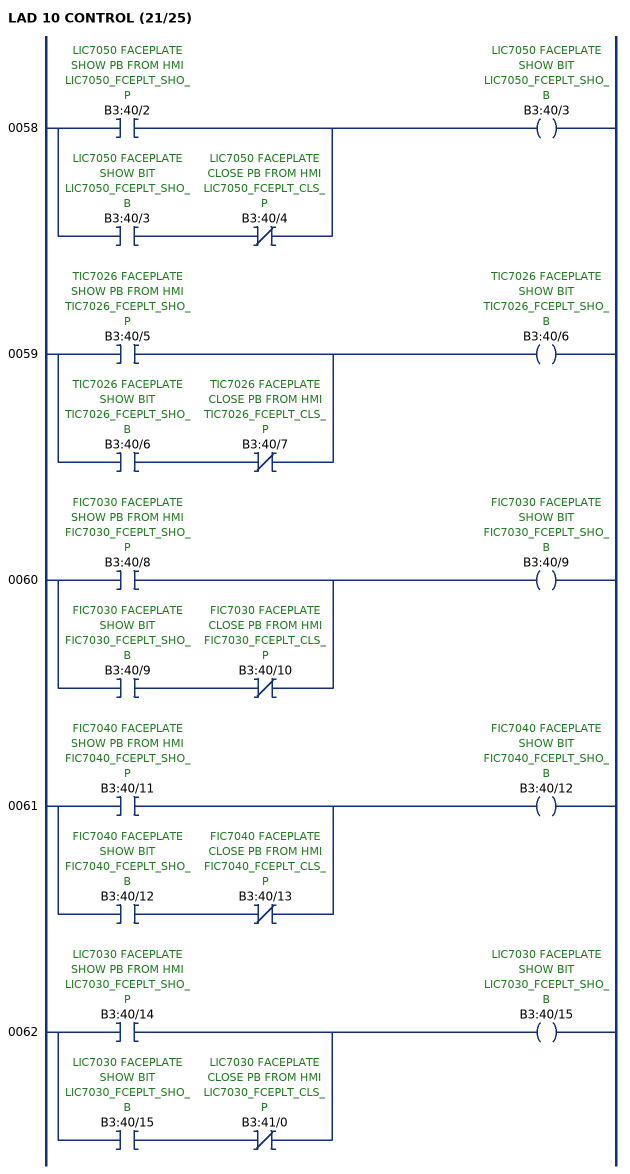
% Rung: 58 %
SOR BST XIC B3:40/2 NXB XIC B3:40/3 XIO B3:40/4 BND OTE B3:40/3 EOR
%   B3:40/2  LIC7050_FCEPLT_SHO_P  "LIC7050 FACEPLATE SHOW PB FROM HMI" %
%   B3:40/3  LIC7050_FCEPLT_SHO_B  "LIC7050 FACEPLATE SHOW BIT" %
%   B3:40/4  LIC7050_FCEPLT_CLS_P  "LIC7050 FACEPLATE CLOSE PB FROM HMI" %
% Rung: 59 %
SOR BST XIC B3:40/5 NXB XIC B3:40/6 XIO B3:40/7 BND OTE B3:40/6 EOR
%   B3:40/5  TIC7026_FCEPLT_SHO_P  "TIC7026 FACEPLATE SHOW PB FROM HMI" %
%   B3:40/6  TIC7026_FCEPLT_SHO_B  "TIC7026 FACEPLATE SHOW BIT" %
%   B3:40/7  TIC7026_FCEPLT_CLS_P  "TIC7026 FACEPLATE CLOSE PB FROM HMI" %
% Rung: 60 %
SOR BST XIC B3:40/8 NXB XIC B3:40/9 XIO B3:40/10 BND OTE B3:40/9 EOR
%   B3:40/8  FIC7030_FCEPLT_SHO_P  "FIC7030 FACEPLATE SHOW PB FROM HMI" %
%   B3:40/9  FIC7030_FCEPLT_SHO_B  "FIC7030 FACEPLATE SHOW BIT" %
%   B3:40/10  FIC7030_FCEPLT_CLS_P  "FIC7030 FACEPLATE CLOSE PB FROM HMI" %
% Rung: 61 %
SOR BST XIC B3:40/11 NXB XIC B3:40/12 XIO B3:40/13 BND OTE B3:40/12 EOR
%   B3:40/11  FIC7040_FCEPLT_SHO_P  "FIC7040 FACEPLATE SHOW PB FROM HMI" %
%   B3:40/12  FIC7040_FCEPLT_SHO_B  "FIC7040 FACEPLATE SHOW BIT" %
%   B3:40/13  FIC7040_FCEPLT_CLS_P  "FIC7040 FACEPLATE CLOSE PB FROM HMI" %
% Rung: 62 %
SOR BST XIC B3:40/14 NXB XIC B3:40/15 XIO B3:41/0 BND OTE B3:40/15 EOR
%   B3:40/14  LIC7030_FCEPLT_SHO_P  "LIC7030 FACEPLATE SHOW PB FROM HMI" %
%   B3:40/15  LIC7030_FCEPLT_SHO_B  "LIC7030 FACEPLATE SHOW BIT" %
%   B3:41/0  LIC7030_FCEPLT_CLS_P  "LIC7030 FACEPLATE CLOSE PB FROM HMI" %

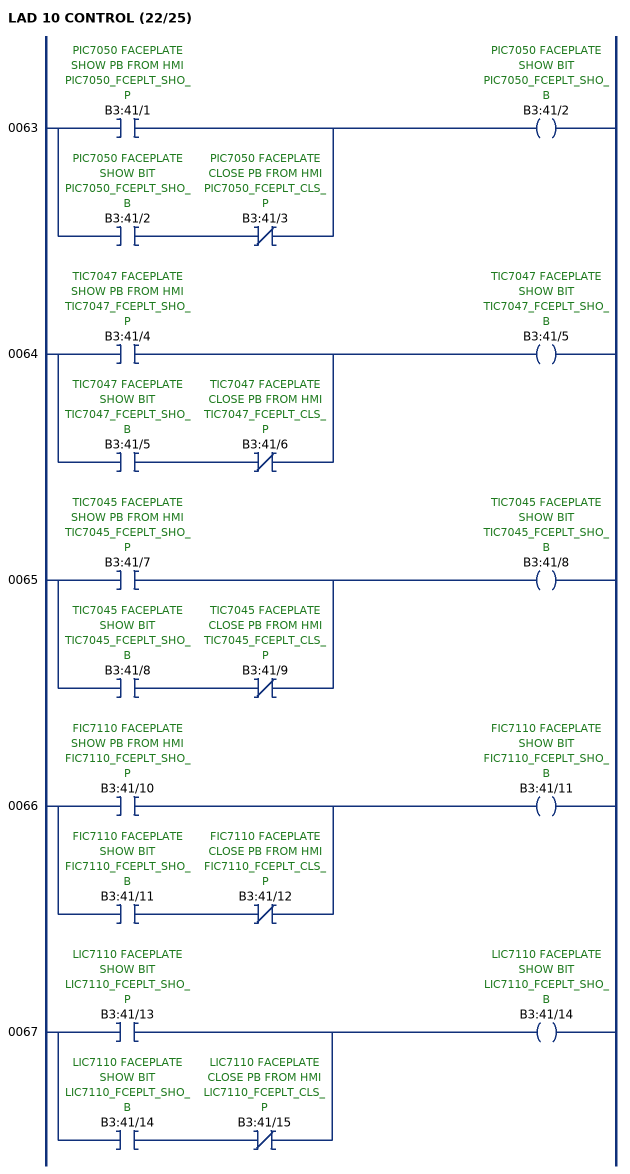
% Rung: 63 %
SOR BST XIC B3:41/1 NXB XIC B3:41/2 XIO B3:41/3 BND OTE B3:41/2 EOR
%   B3:41/1  PIC7050_FCEPLT_SHO_P  "PIC7050 FACEPLATE SHOW PB FROM HMI" %
%   B3:41/2  PIC7050_FCEPLT_SHO_B  "PIC7050 FACEPLATE SHOW BIT" %
%   B3:41/3  PIC7050_FCEPLT_CLS_P  "PIC7050 FACEPLATE CLOSE PB FROM HMI" %
% Rung: 64 %
SOR BST XIC B3:41/4 NXB XIC B3:41/5 XIO B3:41/6 BND OTE B3:41/5 EOR
%   B3:41/4  TIC7047_FCEPLT_SHO_P  "TIC7047 FACEPLATE SHOW PB FROM HMI" %
%   B3:41/5  TIC7047_FCEPLT_SHO_B  "TIC7047 FACEPLATE SHOW BIT" %
%   B3:41/6  TIC7047_FCEPLT_CLS_P  "TIC7047 FACEPLATE CLOSE PB FROM HMI" %
% Rung: 65 %
SOR BST XIC B3:41/7 NXB XIC B3:41/8 XIO B3:41/9 BND OTE B3:41/8 EOR
%   B3:41/7  TIC7045_FCEPLT_SHO_P  "TIC7045 FACEPLATE SHOW PB FROM HMI" %
%   B3:41/8  TIC7045_FCEPLT_SHO_B  "TIC7045 FACEPLATE SHOW BIT" %
%   B3:41/9  TIC7045_FCEPLT_CLS_P  "TIC7045 FACEPLATE CLOSE PB FROM HMI" %
% Rung: 66 %
SOR BST XIC B3:41/10 NXB XIC B3:41/11 XIO B3:41/12 BND OTE B3:41/11 EOR
%   B3:41/10  FIC7110_FCEPLT_SHO_P  "FIC7110 FACEPLATE SHOW PB FROM HMI" %
%   B3:41/11  FIC7110_FCEPLT_SHO_B  "FIC7110 FACEPLATE SHOW BIT" %
%   B3:41/12  FIC7110_FCEPLT_CLS_P  "FIC7110 FACEPLATE CLOSE PB FROM HMI" %
% Rung: 67 %
SOR BST XIC B3:41/13 NXB XIC B3:41/14 XIO B3:41/15 BND OTE B3:41/14 EOR
%   B3:41/13  LIC7110_FCEPLT_SHO_P  "LIC7110 FACEPLATE SHOW BIT" %
%   B3:41/14  LIC7110_FCEPLT_SHO_B  "LIC7110 FACEPLATE SHOW BIT" %
%   B3:41/15  LIC7110_FCEPLT_CLS_P  "LIC7110 FACEPLATE CLOSE PB FROM HMI" %

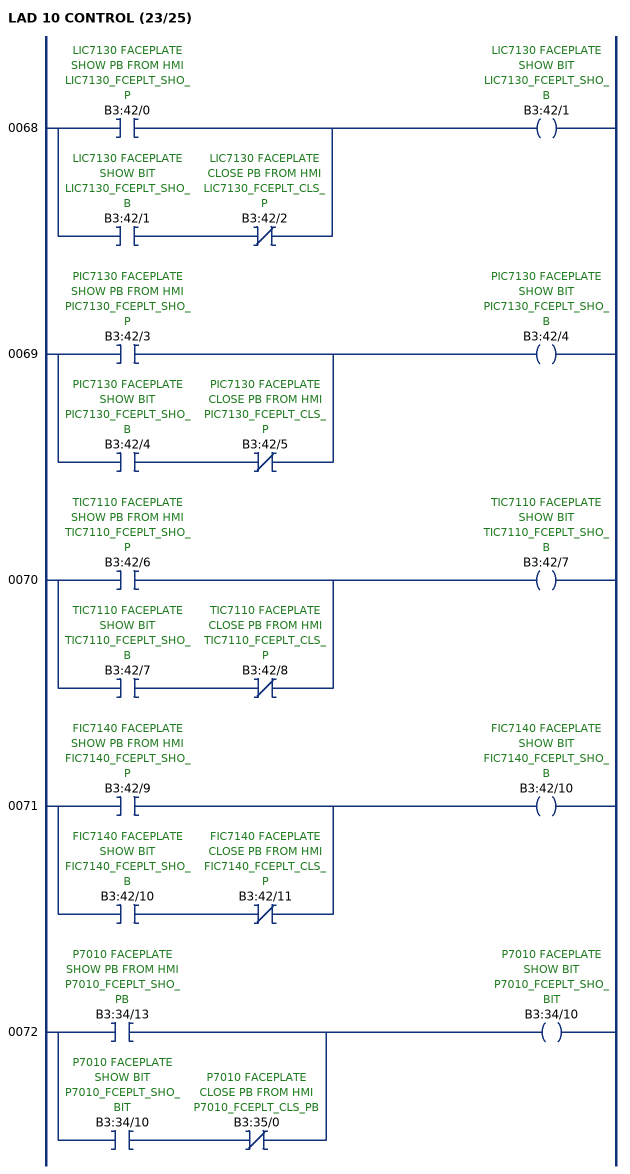
% Rung: 68 %
SOR BST XIC B3:42/0 NXB XIC B3:42/1 XIO B3:42/2 BND OTE B3:42/1 EOR
%   B3:42/0  LIC7130_FCEPLT_SHO_P  "LIC7130 FACEPLATE SHOW PB FROM HMI" %
%   B3:42/1  LIC7130_FCEPLT_SHO_B  "LIC7130 FACEPLATE SHOW BIT" %
%   B3:42/2  LIC7130_FCEPLT_CLS_P  "LIC7130 FACEPLATE CLOSE PB FROM HMI" %
% Rung: 69 %
SOR BST XIC B3:42/3 NXB XIC B3:42/4 XIO B3:42/5 BND OTE B3:42/4 EOR
%   B3:42/3  PIC7130_FCEPLT_SHO_P  "PIC7130 FACEPLATE SHOW PB FROM HMI" %
%   B3:42/4  PIC7130_FCEPLT_SHO_B  "PIC7130 FACEPLATE SHOW BIT" %
%   B3:42/5  PIC7130_FCEPLT_CLS_P  "PIC7130 FACEPLATE CLOSE PB FROM HMI" %
% Rung: 70 %
SOR BST XIC B3:42/6 NXB XIC B3:42/7 XIO B3:42/8 BND OTE B3:42/7 EOR
%   B3:42/6  TIC7110_FCEPLT_SHO_P  "TIC7110 FACEPLATE SHOW PB FROM HMI" %
%   B3:42/7  TIC7110_FCEPLT_SHO_B  "TIC7110 FACEPLATE SHOW BIT" %
%   B3:42/8  TIC7110_FCEPLT_CLS_P  "TIC7110 FACEPLATE CLOSE PB FROM HMI" %
% Rung: 71 %
SOR BST XIC B3:42/9 NXB XIC B3:42/10 XIO B3:42/11 BND OTE B3:42/10 EOR
%   B3:42/9  FIC7140_FCEPLT_SHO_P  "FIC7140 FACEPLATE SHOW PB FROM HMI" %
%   B3:42/10  FIC7140_FCEPLT_SHO_B  "FIC7140 FACEPLATE SHOW BIT" %
%   B3:42/11  FIC7140_FCEPLT_CLS_P  "FIC7140 FACEPLATE CLOSE PB FROM HMI" %
% Rung: 72 %
SOR BST XIC B3:34/13 NXB XIC B3:34/10 XIO B3:35/0 BND OTE B3:34/10 EOR
%   B3:34/13  P7010_FCEPLT_SHO_PB  "P7010 FACEPLATE SHOW PB FROM HMI" %
%   B3:34/10  P7010_FCEPLT_SHO_BIT  "P7010 FACEPLATE SHOW BIT" %
%   B3:35/0  P7010_FCEPLT_CLS_PB  "P7010 FACEPLATE CLOSE PB FROM HMI" %

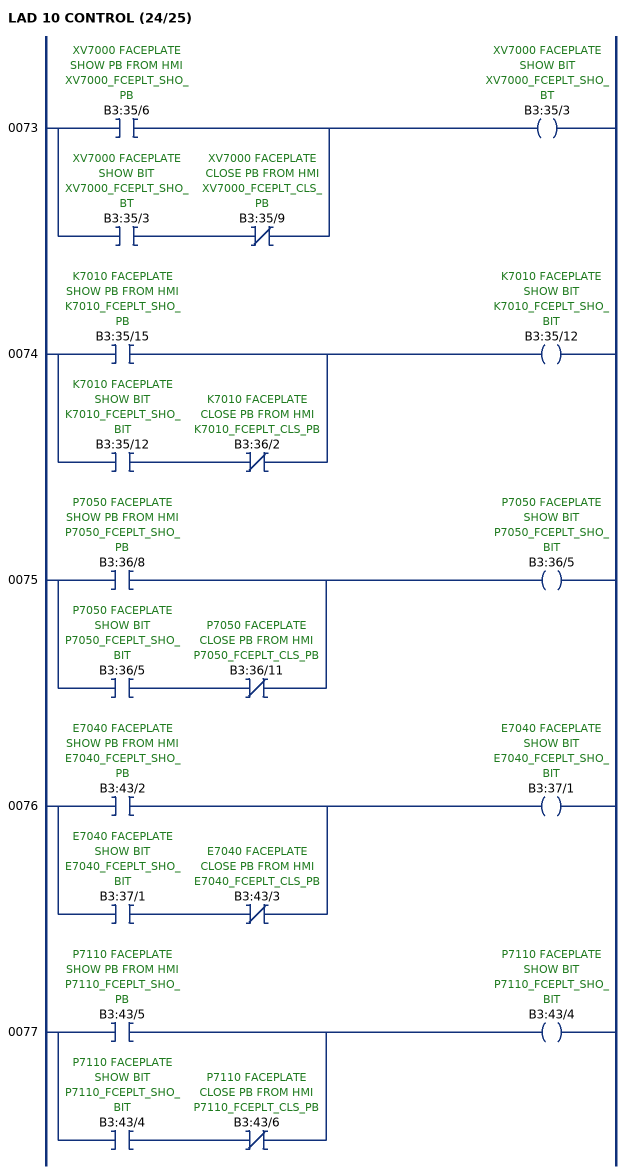
% Rung: 73 %
SOR BST XIC B3:35/6 NXB XIC B3:35/3 XIO B3:35/9 BND OTE B3:35/3 EOR
%   B3:35/6  XV7000_FCEPLT_SHO_PB  "XV7000 FACEPLATE SHOW PB FROM HMI" %
%   B3:35/3  XV7000_FCEPLT_SHO_BT  "XV7000 FACEPLATE SHOW BIT" %
%   B3:35/9  XV7000_FCEPLT_CLS_PB  "XV7000 FACEPLATE CLOSE PB FROM HMI" %
% Rung: 74 %
SOR BST XIC B3:35/15 NXB XIC B3:35/12 XIO B3:36/2 BND OTE B3:35/12 EOR
%   B3:35/15  K7010_FCEPLT_SHO_PB  "K7010 FACEPLATE SHOW PB FROM HMI" %
%   B3:35/12  K7010_FCEPLT_SHO_BIT  "K7010 FACEPLATE SHOW BIT" %
%   B3:36/2  K7010_FCEPLT_CLS_PB  "K7010 FACEPLATE CLOSE PB FROM HMI" %
% Rung: 75 %
SOR BST XIC B3:36/8 NXB XIC B3:36/5 XIO B3:36/11 BND OTE B3:36/5 EOR
%   B3:36/8  P7050_FCEPLT_SHO_PB  "P7050 FACEPLATE SHOW PB FROM HMI" %
%   B3:36/5  P7050_FCEPLT_SHO_BIT  "P7050 FACEPLATE SHOW BIT" %
%   B3:36/11  P7050_FCEPLT_CLS_PB  "P7050 FACEPLATE CLOSE PB FROM HMI" %
% Rung: 76 %
SOR BST XIC B3:43/2 NXB XIC B3:37/1 XIO B3:43/3 BND OTE B3:37/1 EOR
%   B3:43/2  E7040_FCEPLT_SHO_PB  "E7040 FACEPLATE SHOW PB FROM HMI" %
%   B3:37/1  E7040_FCEPLT_SHO_BIT  "E7040 FACEPLATE SHOW BIT" %
%   B3:43/3  E7040_FCEPLT_CLS_PB  "E7040 FACEPLATE CLOSE PB FROM HMI" %
% Rung: 77 %
SOR BST XIC B3:43/5 NXB XIC B3:43/4 XIO B3:43/6 BND OTE B3:43/4 EOR
%   B3:43/5  P7110_FCEPLT_SHO_PB  "P7110 FACEPLATE SHOW PB FROM HMI" %
%   B3:43/4  P7110_FCEPLT_SHO_BIT  "P7110 FACEPLATE SHOW BIT" %
%   B3:43/6  P7110_FCEPLT_CLS_PB  "P7110 FACEPLATE CLOSE PB FROM HMI" %

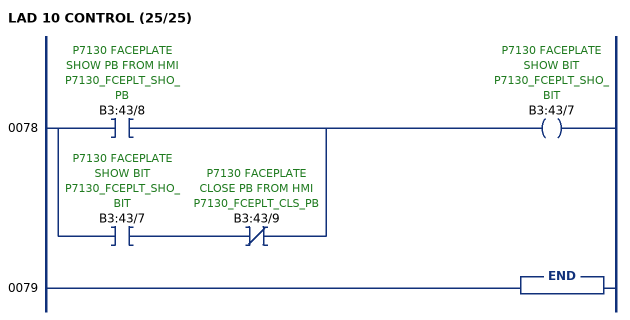
% Rung: 78 %
SOR BST XIC B3:43/8 NXB XIC B3:43/7 XIO B3:43/9 BND OTE B3:43/7 EOR
%   B3:43/8  P7130_FCEPLT_SHO_PB  "P7130 FACEPLATE SHOW PB FROM HMI" %
%   B3:43/7  P7130_FCEPLT_SHO_BIT  "P7130 FACEPLATE SHOW BIT" %
%   B3:43/9  P7130_FCEPLT_CLS_PB  "P7130 FACEPLATE CLOSE PB FROM HMI" %
% Rung: 79 %
SOR END EOR

OTHER DOCUMENTED ADDRESSES
  B3:46/11  "DUMMY"
  B3:47/0  "ONE SHOT"
  B3:47/1  "ONE SHOT"
  B3:47/2  "ONE SHOT"
  B3:47/3  "ONE SHOT"
  B3:47/4  "ONE SHOT"
  B3:47/5  "ONE SHOT"
  B3:47/6  "ONE SHOT"
  B3:47/7  "ONE SHOT"
  B3:47/8  "ONE SHOT"
  B3:47/9  "ONE SHOT"
  B3:47/10  "ONE SHOT"
  B3:47/11  "ONE SHOT"
  B3:47/12  "ONE SHOT"
  B3:47/13  "ONE SHOT"
  B3:47/14  "ONE SHOT"
  B3:47/15  "ONE SHOT"
  B3:48/0  "ONE SHOT"
  B3:48/1  "ONE SHOT"
  B3:48/2  "ONE SHOT"
  B9:36/2  "ESD LIC-7130 OFF"
  DFILE:0  "OUTPUT"
  DFILE:1  "INPUT"
  DFILE:2  "STATUS"
  DFILE:3  "BINARY"
  DFILE:4  "TIMER"
  DFILE:5  "COUNTER"
  DFILE:6  "CONTROL"
  DFILE:7  "INTEGER"
  DFILE:8  "FLOAT"
  DFILE:9  "ALARMS"
  DFILE:10  "F-SETPTS 1"
  DFILE:11  "N-SETPTS 1"
  DFILE:12  "PIDBLOCKS1"
  DFILE:13  "DONOTTOUCH"
  DFILE:14  "PIDBLOCKS2"
  DFILE:15  "PIDBLOCKS3"
  DFILE:16  "SYSCTRLS"
  DFILE:17  "TIMERS 2"
  DFILE:18  "F-SETPTS 2"
  DFILE:19  "N-SETPTS 2"
  DFILE:20  "MB_CFG"
  DFILE:21  "MB_BIN"
  DFILE:22  "MB_FLT1"
  DFILE:23  "MB_FLT2"
  DFILE:24  "MB_FLT3"
  DFILE:25  "MB_FLT4"
  DFILE:26  "MB_FLT5"
  DFILE:27  "MB_FLT6"
  DFILE:28  "MB_FLT7"
  DFILE:29  "COMP_4"
  F10:[N7:100]  F18
  F22:0  FT_7002_SCI_PLC  "FT-7002 Scaled In 0-600 PLC -> DeltaV"
  F22:1  FT_7010_SCI_PLC  "FT-7010 Scaled In 0-200 PLC -> DeltaV"
  F22:2  LT_7010_SCI_PLC  "LT-7010 Scaled In 0-100 PLC -> DeltaV"
  F22:3  PT_7010_SCI_PLC  "PT-7010 Scaled In 0-200 PLC -> DeltaV"
  F22:4  PT_7020_SCI_PLC  "PT-7020 Scaled In 0-1000 PLC -> DeltaV"
  F22:5  FT_7000_SCI_PLC  "FT-7000 Scaled In 0-40 PLC -> DeltaV"
  F22:6  FT_7005_SCI_PLC  "FT-7005 Scaled In 0-300 PLC -> DeltaV"
  F22:7  FT_7008_SCI_PLC  "FT-7008 Scaled In 0-500 PLC -> DeltaV"
  F22:8  FT_7025_SCI_PLC  "FT-7025 Scaled In 0-200 PLC -> DeltaV"
  F22:9  FT_7050_SCI_PLC  "FT-7050 Scaled In 0-150 PLC -> DeltaV"
  F22:10  LT_7050_SCI_PLC  "LT-7050 Scaled In 0-100 PLC -> DeltaV"
  F22:11  PT_7000_SCI_PLC  "PT-7000 Scaled In 0-1000 PLC -> DeltaV"
  F22:12  PT_7015_SCI_PLC  "PT-7015 Scaled In 0-1000 PLC -> DeltaV"
  F22:13  PT_7025_SCI_PLC  "PT-7025 Scaled In 0-1000 PLC -> DeltaV"
  F22:14  FT_7030_SCI_PLC  "FT-7030 Scaled In 0-200 PLC -> DeltaV"
  F22:15  FT_7040_SCI_PLC  "FT-7040 Scaled In 0-50 PLC -> DeltaV"
  F22:16  FT_7052_SCI_PLC  "FT-7052 Scaled In 0-150 PLC -> DeltaV"
  F22:17  LT_7030_SCI_PLC  "LT-7030 Scaled In 0-100 PLC -> DeltaV"
  F22:18  PDT_7040_SCI_PLC  "PDT-7040 Scaled In 0-5 PLC -> DeltaV"
  F22:19  PT_7030_SCI_PLC  "PT-7030 Scaled In 0-1000 PLC -> DeltaV"
  F22:20  PT_7040_SCI_PLC  "PT-7040 Scaled In 0-1000 PLC -> DeltaV"
  F22:21  PT_7050_SCI_PLC  "PT-7050 Scaled In 0-1000 PLC -> DeltaV"
  F22:22  ST_7040_SCI_PLC  "ST-7040 Scaled In 0-100 PLC -> DeltaV"
  F22:23  FT_7095_SCI_PLC  "FT-7095 Scaled In 0-700 PLC -> DeltaV"
  F22:24  FT_7110_SCI_PLC  "FT-7110 Scaled In 0-400 PLC -> DeltaV"
  F22:25  FT_7130_SCI_PLC  "FT-7130 Scaled In 0-3 PLC -> DeltaV"
  F22:26  FT_7132_SCI_PLC  "FT-7132 Scaled In 0-700 PLC -> DeltaV"
  F22:27  FT_7145_SCI_PLC  "FT-7145 Scaled In 0-400 PLC -> DeltaV"
  F22:28  LT_7110_SCI_PLC  "LT-7110 Scaled In 0-100 PLC -> DeltaV"
  F22:29  LT_7130_SCI_PLC  "LT-7130 Scaled In 0-100 PLC -> DeltaV"
  F22:30  PDT_7110_SCI_PLC  "PDT-7110 Scaled In 0-5 PLC -> DeltaV"
  F22:31  PT_7110_SCI_PLC  "PT-7110 Scaled In 0-300 PLC -> DeltaV"
  F22:32  PT_7111_SCI_PLC  "PT-7111 Scaled In 0-200 PLC -> DeltaV"
  F22:33  PT_7130_SCI_PLC  "PT-7130 Scaled In 0-200 PLC -> DeltaV"
  F22:34  ST_7110_SCI_PLC  "ST-7110 Scaled In 0-100 PLC -> DeltaV"
  F22:35  ST_7130_SCI_PLC  "ST-7130 Scaled In 0-100 PLC -> DeltaV"
  F22:36  FT_7120_SCI_PLC  "FT-7120 Scaled In 0-400 PLC -> DeltaV"
  F22:37  FT_7140_SCI_PLC  "FT-7140 Scaled In (-454-2498) PLC -> DeltaV"
  F22:38  TT_7009_SCI_PLC  "TT-7009 Scaled In (-454-2498) PLC -> DeltaV"
  F22:39  TT_7010_SCI_PLC  "TT-7010 Scaled In (-454-2498) PLC -> DeltaV"
  F22:40  TT_7020_SCI_PLC  "TT-7020 Scaled In (-454-2498) PLC -> DeltaV"
  F22:41  TT_7000_SCI_PLC  "TT-7000 Scaled In (-454-2498) PLC -> DeltaV"
  F22:42  TT_7015_SCI_PLC  "TT-7015 Scaled In (-454-2498) PLC -> DeltaV"
  F22:43  TT_7025_SCI_PLC  "TT-7025 Scaled In (-454-2498) PLC -> DeltaV"
  F22:44  TT_7026_SCI_PLC  "TT-7026 Scaled In (-454-2498) PLC -> DeltaV"
  F22:45  TT_7050_SCI_PLC  "TT-7050 Scaled In (-454-2498) PLC -> DeltaV"
  F22:46  TT_7030_SCI_PLC  "TT-7030 Scaled In (-454-2498) PLC -> DeltaV"
  F22:47  TT_7040_SCI_PLC  "TT-7040 Scaled In (-454-2498) PLC -> DeltaV"
  F22:48  TT_7042_SCI_PLC  "TT-7042 Scaled In (-454-2498) PLC -> DeltaV"
  F22:49  TT_7043_SCI_PLC  "TT-7043 Scaled In (-454-2498) PLC -> DeltaV"
  F22:50  TT_7044_SCI_PLC  "TT-7044 Scaled In (-454-2498) PLC -> DeltaV"
  F22:51  TT_7045_SCI_PLC  "TT-7045 Scaled In (-454-2498) PLC -> DeltaV"
  F22:52  TT_7046_SCI_PLC  "TT-7046 Scaled In (-454-2498) PLC -> DeltaV"
  F22:53  TT_7047_SCI_PLC  "TT-7047 Scaled In (-454-2498) PLC -> DeltaV"
  F22:54  TT_7110_SCI_PLC  "TT-7110 Scaled In (-454-2498) PLC -> DeltaV"
  F22:55  TT_7111_SCI_PLC  "TT-7111 Scaled In (-454-2498) PLC -> DeltaV"
  F22:56  TT_7118_SCI_PLC  "TT-7118 Scaled In (-454-2498) PLC -> DeltaV"
  F22:57  TT_7119_SCI_PLC  "TT-7119 Scaled In (-454-2498) PLC -> DeltaV"
  F22:58  TT_7130_SCI_PLC  "TT-7130 Scaled In (-454-2498) PLC -> DeltaV"
  F22:59  ST_7010_SCI_PLC  "ST-7010 Scaled In 0-100 PLC -> DeltaV"
  F22:60  TT_7135_SCI_PLC  "TT-7135 Scaled In (-454-2498) PLC -> DeltaV"
  F22:61  TT_7140_SCI_PLC  "TT-7140 Scaled In (-454-2498) PLC -> DeltaV"
  F22:62  TT_7145_SCI_PLC  "TT-7145 Scaled In (-454-2498) PLC -> DeltaV"
  F22:63  PT_7026_SCI_PLC  "PT-7026 Scaled In 0-1000 PLC -> DeltaV"
  F22:64  TT_7027_SCI_PLC  "TT-7027 Scaled In (-454-2498) PLC -> DeltaV"
  F22:65  FIC7015_PV_PLC  "FIC7015 PV SCALED FOR HMI PLC -> DeltaV"
  F22:66  TIC7010_PV_PLC  "TIC7010 PV SCALED FOR HMI PLC -> DeltaV"
  F22:67  FIC7000_PV_PLC  "FIC7000 PV SCALED FOR HMI PLC -> DeltaV"
  F22:68  FIC7005_PV_PLC  "FIC7005 PV SCALED FOR HMI PLC -> DeltaV"
  F22:69  FIC7008_PV_PLC  "FIC7008 PV SCALED FOR HMI PLC -> DeltaV"
  F22:70  FIC7010_PV_PLC  "FIC7010 PV SCALED FOR HMI PLC -> DeltaV"
  F22:71  LIC7050_PV_PLC  "LIC7050 PV SCALED FOR HMI PLC -> DeltaV"
  F22:72  TIC7026_PV_PLC  "TIC7026 PV SCALED FOR HMI PLC -> DeltaV"
  F22:73  FIC7030_PV_PLC  "FIC7030 PV SCALED FOR HMI PLC -> DeltaV"
  F22:74  FIC7040_PV_PLC  "FIC7040 PV SCALED FOR HMI PLC -> DeltaV"
  F22:75  LIC7030_PV_PLC  "LIC7030 PV SCALED FOR HMI PLC -> DeltaV"
  F22:76  PIC7050_PV_PLC  "PIC7050 PV SCALED FOR HMI PLC -> DeltaV"
  F22:77  TIC7047_PV_PLC  "TIC7047 PV SCALED FOR HMI PLC -> DeltaV"
  F22:78  TIC7045_PV_PLC  "TIC7045 PV SCALED FOR HMI PLC -> DeltaV"
  F22:79  FIC7110_PV_PLC  "FIC7110 PV SCALED FOR HMI PLC -> DeltaV"
  F22:80  LIC7110_PV_PLC  "LIC7110 PV SCALED FOR HMI PLC -> DeltaV"
  F22:81  LIC7130_PV_PLC  "LIC7130 PV SCALED FOR HMI PLC -> DeltaV"
  F22:82  PIC7130_PV_PLC  "PIC7130 PV SCALED FOR HMI PLC -> DeltaV"
  F22:83  TIC7110_PV_PLC  "TIC7110 PV SCALED FOR HMI PLC -> DeltaV"
  F22:84  FIC7140_PV_PLC  "FIC7140 PV SCALED FOR HMI PLC -> DeltaV"
  F22:85  WATCHDOG_TIMER_PLC  "PLC WATCHDOG TIMER PLC -> DeltaV"
  F23:0  FT_7002_L_AL_SP_PLC  "FT-7002 LO ALARM SP PLC -> DeltaV"
  F23:1  FT_7002_H_AL_SP_PLC  "FT-7002 HI ALARM SP PLC -> DeltaV"
  F23:2  FT_7010_L_AL_SP_PLC  "FT-7010 LO ALARM SP PLC -> DeltaV"
  F23:3  FT_7010_H_AL_SP_PLC  "FT-7010 HI ALARM SP PLC -> DeltaV"
  F23:4  LT_7010_L_AL_SP_PLC  "LT-7010 LO ALARM SP PLC -> DeltaV"
  F23:5  LT_7010_H_AL_SP_PLC  "LT-7010 HI ALARM SP PLC -> DeltaV"
  F23:6  PT_7010_L_AL_SP_PLC  "PT-7010 LO ALARM SP PLC -> DeltaV"
  F23:7  PT_7010_H_AL_SP_PLC  "PT-7010 HI ALARM SP PLC -> DeltaV"
  F23:8  PT_7020_L_AL_SP_PLC  "PT-7020 LO ALARM SP PLC -> DeltaV"
  F23:9  PT_7020_H_AL_SP_PLC  "PT-7020 HI ALARM SP PLC -> DeltaV"
  F23:10  FT_7000_L_AL_SP_PLC  "FT-7000 LO ALARM SP PLC -> DeltaV"
  F23:11  FT_7000_H_AL_SP_PLC  "FT-7000 HI ALARM SP PLC -> DeltaV"
  F23:12  FT_7005_L_AL_SP_PLC  "FT-7005 LO ALARM SP PLC -> DeltaV"
  F23:13  FT_7005_H_AL_SP_PLC  "FT-7005 HI ALARM SP PLC -> DeltaV"
  F23:14  FT_7008_L_AL_SP_PLC  "FT-7008 LO ALARM SP PLC -> DeltaV"
  F23:15  FT_7008_H_AL_SP_PLC  "FT-7008 HI ALARM SP PLC -> DeltaV"
  F23:16  FT_7025_L_AL_SP_PLC  "FT-7025 LO ALARM SP PLC -> DeltaV"
  F23:17  FT_7025_H_AL_SP_PLC  "FT-7025 HI ALARM SP PLC -> DeltaV"
  F23:18  FT_7050_L_AL_SP_PLC  "FT-7050 LO ALARM SP PLC -> DeltaV"
  F23:19  FT_7050_H_AL_SP_PLC  "FT-7050 HI ALARM SP PLC -> DeltaV"
  F23:20  LT_7050_L_AL_SP_PLC  "LT-7050 LO ALARM SP PLC -> DeltaV"
  F23:21  LT_7050_H_AL_SP_PLC  "LT-7050 HI ALARM SP PLC -> DeltaV"
  F23:22  PT_7000_L_AL_SP_PLC  "PT-7000 LO ALARM SP PLC -> DeltaV"
  F23:23  PT_7000_H_AL_SP_PLC  "PT-7000 HI ALARM SP PLC -> DeltaV"
  F23:24  PT_7015_L_AL_SP_PLC  "PT-7015 LO ALARM SP PLC -> DeltaV"
  F23:25  PT_7015_H_AL_SP_PLC  "PT-7015 HI ALARM SP PLC -> DeltaV"
  F23:26  PT_7025_L_AL_SP_PLC  "PT-7025 LO ALARM SP PLC -> DeltaV"
  F23:27  PT_7025_H_AL_SP_PLC  "PT-7025 HI ALARM SP PLC -> DeltaV"
  F23:28  FT_7030_L_AL_SP_PLC  "FT-7030 LO ALARM SP PLC -> DeltaV"
  F23:29  FT_7030_H_AL_SP_PLC  "FT-7030 HI ALARM SP PLC -> DeltaV"
  F23:30  FT_7040_L_ALSP_PLC  "FT-7040 LO ALARM SP PLC -> DeltaV"
  F23:31  FT_7040_H_AL_SP_PLC  "FT-7040 HI ALARM SP PLC -> DeltaV"
  F23:32  FT_7052_L_AL_SP_PLC  "FT-7052 LO ALARM SP PLC -> DeltaV"
  F23:33  FT_7052_H_AL_SP_PLC  "FT-7052 HI ALARM SP PLC -> DeltaV"
  F23:34  LT_7030_L_AL_SP_PLC  "LT-7030 LO ALARM SP PLC -> DeltaV"
  F23:35  LT_7030_H_AL_SP_PLC  "LT-7030 HI ALARM SP PLC -> DeltaV"
  F23:36  PDT_7040_L_AL_SP_PLC  "PDT-7040 LO ALARM SP PLC -> DeltaV"
  F23:37  PDT_7040_H_AL_SP_PLC  "PDT-7040 HI ALARM SP PLC -> DeltaV"
  F23:38  PT_7030_L_AL_SP_PLC  "PT-7030 LO ALARM SP PLC -> DeltaV"
  F23:39  PT_7030_H_AL_SP_PLC  "PT-7030 HI ALARM SP PLC -> DeltaV"
  F23:40  PT_7040_L_AL_SP_PLC  "PT-7040 LO ALARM SP PLC -> DeltaV"
  F23:41  PT_7040_H_AL_SP_PLC  "PT-7040 HI ALARM SP PLC -> DeltaV"
  F23:42  PT_7050_L_AL_SP_PLC  "PT-7050 LO ALARM SP PLC -> DeltaV"
  F23:43  PT_7050_H_AL_SP_PLC  "PT-7050 HI ALARM SP PLC -> DeltaV"
  F23:44  ST_7040_L_AL_SP_PLC  "ST-7040 LO ALARM SP PLC -> DeltaV"
  F23:45  ST_7040_H_AL_SP_PLC  "ST-7040 HI ALARM SP PLC -> DeltaV"
  F23:46  FT_7095_L_AL_SP_PLC  "FT-7095 LO ALARM SP PLC -> DeltaV"
  F23:47  FT_7095_H_AL_SP_PLC  "FT-7095 HI ALARM SP PLC -> DeltaV"
  F23:48  FT_7110_L_AL_SP_PLC  "FT-7110 LO ALARM SP PLC -> DeltaV"
  F23:49  FT_7110_H_AL_SP_PLC  "FT-7110 HI ALARM SP PLC -> DeltaV"
  F23:50  FT_7130_L_AL_SP_PLC  "FT-7130 LO ALARM SP PLC -> DeltaV"
  F23:51  FT_7130_H_AL_SP_PLC  "FT-7130 HI ALARM SP PLC -> DeltaV"
  F23:52  FT_7132_L_AL_SP_PLC  "FT-7132 LO ALARM SP PLC -> DeltaV"
  F23:53  FT_7132_H_AL_SP_PLC  "FT-7132 HI ALARM SP PLC -> DeltaV"
  F23:54  FT_7145_L_AL_SP_PLC  "FT-7145 LO ALARM SP PLC -> DeltaV"
  F23:55  FT_7145_H_AL_SP_PLC  "FT-7145 HI ALARM SP PLC -> DeltaV"
  F23:56  LT_7110_L_AL_SP_PLC  "LT-7110 LO ALARM SP PLC -> DeltaV"
  F23:57  LT_7110_H_AL_SP_PLC  "LT-7110 HI ALARM SP PLC -> DeltaV"
  F23:58  LT_7130_L_AL_SP_PLC  "LT-7130 LO ALARM SP PLC -> DeltaV"
  F23:59  LT_7130_H_AL_SP_PLC  "LT-7130 HI ALARM SP PLC -> DeltaV"
  F23:60  PDT7110_L_AL_SP_PLC  "PDT-7110 LO ALARM SP PLC -> DeltaV"
  F23:61  PDT7110_H_AL_SP_PLC  "PDT-7110 HI ALARM SP PLC -> DeltaV"
  F23:62  PT_7110_L_AL_SP_PLC  "PT-7110 LO ALARM SP PLC -> DeltaV"
  F23:63  PT_7110_H_AL_SP_PLC  "PT-7110 HI ALARM SP PLC -> DeltaV"
  F23:64  PT_7111_L_AL_SP_PLC  "PT-7111 LO ALARM SP PLC -> DeltaV"
  F23:65  PT_7111_H_AL_SP_PLC  "PT-7111 HI ALARM SP PLC -> DeltaV"
  F23:66  PT_7130_L_AL_SP_PLC  "PT-7130 LO ALARM SP PLC -> DeltaV"
  F23:67  PT_7130_H_AL_SP_PLC  "PT-7130 HI ALARM SP PLC -> DeltaV"
  F23:68  ST_7110_L_AL_SP_PLC  "ST-7110 LO ALARM SP PLC -> DeltaV"
  F23:69  ST_7110_H_AL_SP_PLC  "ST-7110 HI ALARM SP PLC -> DeltaV"
  F23:70  ST_7130_L_AL_SP_PLC  "ST-7130 LO ALARM SP PLC -> DeltaV"
  F23:71  ST_7130_H_AL_SP_PLC  "ST-7130 HI ALARM SP PLC -> DeltaV"
  F23:72  FT_7120_L_AL_SP_PLC  "FT-7120 LO ALARM SP PLC -> DeltaV"
  F23:73  FT_7120_H_AL_SP_PLC  "FT-7120 HI ALARM SP PLC -> DeltaV"
  F23:74  FT_7140_L_AL_SP_PLC  "FT-7140 LO ALARM SP PLC -> DeltaV"
  F23:75  FT_7140_H_AL_SP_PLC  "FT-7140 HI ALARM SP PLC -> DeltaV"
  F23:76  TT_7009_L_AL_SP_PLC  "TT-7009 LO ALARM SP PLC -> DeltaV"
  F23:77  TT_7009_H_AL_SP_PLC  "TT-7009 HI ALARM SP PLC -> DeltaV"
  F23:78  TT_7010_L_AL_SP_PLC  "TT-7010 LO ALARM SP PLC -> DeltaV"
  F23:79  TT_7010_H_AL_SP_PLC  "TT-7010 HI ALARM SP PLC -> DeltaV"
  F23:80  TT_7020_L_AL_SP_PLC  "TT-7020 LO ALARM SP PLC -> DeltaV"
  F23:81  TT_7020_H_AL_SP_PLC  "TT-7020 HI ALARM SP PLC -> DeltaV"
  F23:82  TT_7000_L_AL_SP_PLC  "TT-7000 LO ALARM SP PLC -> DeltaV"
  F23:83  TT_7000_H_AL_SP_PLC  "TT-7000 HI ALARM SP PLC -> DeltaV"
  F23:84  TT_7015_L_AL_SP_PLC  "TT-7015 LO ALARM SP PLC -> DeltaV"
  F23:85  TT_7015_H_AL_SP_PLC  "TT-7015 HI ALARM SP PLC -> DeltaV"
  F23:86  TT_7025_L_AL_SP_PLC  "TT-7025 LO ALARM SP PLC -> DeltaV"
  F23:87  TT_7025_H_AL_SP_PLC  "TT-7025 HI ALARM SP PLC -> DeltaV"
  F23:88  TT_7026_L_AL_SP_PLC  "TT-7026 LO ALARM SP PLC -> DeltaV"
  F23:89  TT_7026_H_AL_SP_PLC  "TT-7026 HI ALARM SP PLC -> DeltaV"
  F23:90  TT_7050_L_AL_SP_PLC  "TT-7050 LO ALARM SP PLC -> DeltaV"
  F23:91  TT_7050_H_AL_SP_PLC  "TT-7050 HI ALARM SP PLC -> DeltaV"
  F23:92  TT_7030_L_AL_SP_PLC  "TT-7030 LO ALARM SP PLC -> DeltaV"
  F23:93  TT_7030_H_AL_SP_PLC  "TT-7030 HI ALARM SP PLC -> DeltaV"
  F23:94  TT_7040_L_AL_SP_PLC  "TT-7040 LO ALARM SP PLC -> DeltaV"
  F23:95  TT_7040_H_AL_SP_PLC  "TT-7040 HI ALARM SP PLC -> DeltaV"
  F23:96  TT_7042_L_AL_SP_PLC  "TT-7042 LO ALARM SP PLC -> DeltaV"
  F23:97  TT_7042_H_AL_SP_PLC  "TT-7042 HI ALARM SP PLC -> DeltaV"
  F23:98  TT_7043_L_AL_SP_PLC  "TT-7043L LO ALARM SP PLC -> DeltaV"
  F23:99  TT_7043_H_AL_SP_PLC  "TT-7043L HI ALARM SP PLC -> DeltaV"
  F23:100  TT_7044_L_AL_SP_PLC  "TT-7043R LO ALARM SP PLC -> DeltaV"
  F23:101  TT_7044_H_AL_SP_PLC  "TT-7043R HI ALARM SP PLC -> DeltaV"
  F23:102  TT_7045_L_AL_SP_PLC  "TT-7045 LO ALARM SP PLC -> DeltaV"
  F23:103  TT_7045_H_AL_SP_PLC  "TT-7045 HI ALARM SP PLC -> DeltaV"
  F23:104  TT_7046_L_AL_SP_PLC  "TT-7046 LO ALARM SP PLC -> DeltaV"
  F23:105  TT_7046_H_AL_SP_PLC  "TT-7046 HI ALARM SP PLC -> DeltaV"
  F23:106  TT_7047_L_AL_SP_PLC  "TT-7047 LO ALARM SP PLC -> DeltaV"
  F23:107  TT_7047_H_AL_SP_PLC  "TT-7047 HI ALARM SP PLC -> DeltaV"
  F23:108  TT_7110_L_AL_SP_PLC  "TT-7110 LO ALARM SP PLC -> DeltaV"
  F23:109  TT_7110_H_AL_SP_PLC  "TT-7110 HI ALARM SP PLC -> DeltaV"
  F23:110  TT_7111_L_AL_SP_PLC  "TT-7111 LO ALARM SP PLC -> DeltaV"
  F23:111  TT_7111_H_AL_SP_PLC  "TT-7111 HI ALARM SP PLC -> DeltaV"
  F23:112  TT_7118_L_AL_SP_PLC  "TT-7118 LO ALARM SP PLC -> DeltaV"
  F23:113  TT_7118_H_AL_SP_PLC  "TT-7118 HI ALARM SP PLC -> DeltaV"
  F23:114  TT_7119_L_AL_SP_PLC  "TT-7119 LO ALARM SP PLC -> DeltaV"
  F23:115  TT_7119_H_AL_SP_PLC  "TT-7119 HI ALARM SP PLC -> DeltaV"
  F23:116  TT_7130_L_AL_SP_PLC  "TT-7130 LO ALARM SP PLC -> DeltaV"
  F23:117  TT_7130_H_AL_SP_PLC  "TT-7130 HI ALARM SP PLC -> DeltaV"
  F23:118  ST_7010_LL_SP_PLC  "ST-7010 LOLO ALARM SP PLC -> DeltaV"
  F23:119  ST_7010_L_AL_SP_PLC  "ST-7010 LO ALARM SP PLC -> DeltaV"
  F23:120  TT_7135_L_AL_SP_PLC  "TT-7135 LO ALARM SP PLC -> DeltaV"
  F23:121  TT_7135_H_AL_SP_PLC  "TT-7135 HI ALARM SP PLC -> DeltaV"
  F23:122  TT_7140_L_AL_SP_PLC  "TT-7140 LO ALARM SP PLC -> DeltaV"
  F23:123  TT_7140_H_AL_SP_PLC  "TT-7140 HI ALARM SP PLC -> DeltaV"
  F23:124  TT_7145_L_AL_SP_PLC  "TT-7145 LO ALARM SP PLC -> DeltaV"
  F23:125  TT_7145_H_AL_SP_PLC  "TT-7145 HI ALARM SP PLC -> DeltaV"
  F23:126  FT_7002_LL_SP_PLC  "FT-7002 LOLO ALARM SP PLC -> DeltaV"
  F23:127  FT_7002_HH_SP_PLC  "FT-7002 HIHI ALARM SP PLC -> DeltaV"
  F23:128  FT_7010_LL_SP_PLC  "FT-7010 LOLO ALARM SP PLC -> DeltaV"
  F23:129  FT_7010_HH_SP_PLC  "FT-7010 HIHI ALARM SP PLC -> DeltaV"
  F23:130  LT_7010_LL_SP_PLC  "LT-7010 LOLO ALARM SP PLC -> DeltaV"
  F23:131  LT_7010_HH_SP_PLC  "LT-7010 HIHI ALARM SP PLC -> DeltaV"
  F23:132  PT_7010_LL_SP_PLC  "PT-7010 LOLO ALARM SP PLC -> DeltaV"
  F23:133  PT_7010_HH_SP_PLC  "PT-7010 HIHI ALARM SP PLC -> DeltaV"
  F23:134  PT_7020_LL_SP_PLC  "PT-7020 LOLO ALARM SP PLC -> DeltaV"
  F23:135  PT_7020_HH_SP_PLC  "PT-7020 HIHI ALARM SP PLC -> DeltaV"
  F23:136  FT_7000_LL_SP_PLC  "FT-7000 LOLO ALARM SP PLC -> DeltaV"
  F23:137  FT_7000_HH_SP_PLC  "FT-7000 HIHI ALARM SP PLC -> DeltaV"
  F23:138  FT_7005_LL_SP_PLC  "FT-7005 LOLO ALARM SP PLC -> DeltaV"
  F23:139  FT_7005_HH_SP_PLC  "FT-7005 HIHI ALARM SP PLC -> DeltaV"
  F23:140  FT_7008_LL_SP_PLC  "FT-7008 LOLO ALARM SP PLC -> DeltaV"
  F23:141  FT_7008_HH_SP_PLC  "FT-7008 HIHI ALARM SP PLC -> DeltaV"
  F23:142  FT_7025_LL_SP_PLC  "FT-7025 LOLO ALARM SP PLC -> DeltaV"
  F23:143  FT_7025_HH_SP_PLC  "FT-7025 HIHI ALARM SP PLC -> DeltaV"
  F23:144  FT_7050_LL_SP_PLC  "FT-7050 LOLO ALARM SP PLC -> DeltaV"
  F23:145  FT_7050_HH_SP_PLC  "FT-7050 HIHI ALARM SP PLC -> DeltaV"
  F23:146  LT_7050_LL_SP_PLC  "LT-7050 LOLO ALARM SP PLC -> DeltaV"
  F23:147  LT_7050_HH_SP_PLC  "LT-7050 HIHI ALARM SP PLC -> DeltaV"
  F23:148  PT_7000_LL_SP_PLC  "PT-7000 LOLO ALARM SP PLC -> DeltaV"
  F23:149  PT_7000_HH_SP_PLC  "PT-7000 HIHI ALARM SP PLC -> DeltaV"
  F23:150  PT_7015_LL_SP_PLC  "PT-7015 LOLO ALARM SP PLC -> DeltaV"
  F23:151  PT_7015_HH_SP_PLC  "PT-7015 HIHI ALARM SP PLC -> DeltaV"
  F23:152  PT_7025_LL_SP_PLC  "PT-7025 LOLO ALARM SP PLC -> DeltaV"
  F23:153  PT_7025_HH_SP_PLC  "PT-7025 HIHI ALARM SP PLC -> DeltaV"
  F23:154  FT_7030_LL_SP_PLC  "FT-7030 LOLO ALARM SP PLC -> DeltaV"
  F23:155  FT_7030_HH_SP_PLC  "FT-7030 HIHI ALARM SP PLC -> DeltaV"
  F23:156  FT_7040_LL_SP_PLC  "FT-7040 LOLO ALARM SP PLC -> DeltaV"
  F23:157  FT_7040_HH_SP_PLC  "FT-7040 HIHI ALARM SP PLC -> DeltaV"
  F23:158  FT_7052_LL_SP_PLC  "FT-7052 LOLO ALARM SP PLC -> DeltaV"
  F23:159  FT_7052_HH_SP_PLC  "FT-7052 HIHI ALARM SP PLC -> DeltaV"
  F23:160  LT_7030_LL_SP_PLC  "LT-7030 LOLO ALARM SP PLC -> DeltaV"
  F23:161  LT_7030_HH_SP_PLC  "LT-7030 HIHI ALARM SP PLC -> DeltaV"
  F23:162  PDT_7040_LL_SP_PLC  "PDT-7040 LOLO ALARM SP PLC -> DeltaV"
  F23:163  PDT_7040_HH_SP_PLC  "PDT-7040 HIHI ALARM SP PLC -> DeltaV"
  F23:164  PT_7030_LL_SP_PLC  "PT-7030 LOLO ALARM SP PLC -> DeltaV"
  F23:165  PT_7030_HH_SP_PLC  "PT-7030 HIHI ALARM SP PLC -> DeltaV"
  F23:166  PT_7040_LL_SP_PLC  "PT-7040 LOLO ALARM SP PLC -> DeltaV"
  F23:167  PT_7040_HH_SP_PLC  "PT-7040 HIHI ALARM SP PLC -> DeltaV"
  F23:168  PT_7050_LL_SP_PLC  "PT-7050 LOLO ALARM SP PLC -> DeltaV"
  F23:169  PT_7050_HH_SP_PLC  "PT-7050 HIHI ALARM SP PLC -> DeltaV"
  F23:170  ST_7040_LL_SP_PLC  "ST-7040 LOLO ALARM SP PLC -> DeltaV"
  F23:171  ST_7040_HH_SP_PLC  "ST-7040 HIHI ALARM SP PLC -> DeltaV"
  F23:172  FT_7095_LL_SP_PLC  "FT-7095 LOLO ALARM SP PLC -> DeltaV"
  F23:173  FT_7095_HH_SP_PLC  "FT-7095 HIHI ALARM SP PLC -> DeltaV"
  F23:174  FT_7110_LL_SP_PLC  "FT-7110 LOLO ALARM SP PLC -> DeltaV"
  F23:175  FT_7110_HH_SP_PLC  "FT-7110 HIHI ALARM SP PLC -> DeltaV"
  F23:176  FT_7130_LL_SP_PLC  "FT-7130 LOLO ALARM SP PLC -> DeltaV"
  F23:177  FT_7130_HH_SP_PLC  "FT-7130 HIHI ALARM SP PLC -> DeltaV"
  F23:178  FT_7132_LL_SP_PLC  "FT-7132 LOLO ALARM SP PLC -> DeltaV"
  F23:179  FT_7132_HH_SP_PLC  "FT-7132 HIHI ALARM SP PLC -> DeltaV"
  F23:180  FT_7145_LL_SP_PLC  "FT-7145 LOLO ALARM SP PLC -> DeltaV"
  F23:181  FT_7145_HH_SP_PLC  "FT-7145 HIHI ALARM SP PLC -> DeltaV"
  F23:182  LT_7110_LL_SP_PLC  "LT-7110 LOLO ALARM SP PLC -> DeltaV"
  F23:183  LT_7110_HH_SP_PLC  "LT-7110 HIHI ALARM SP PLC -> DeltaV"
  F23:184  LT_7130_LL_SP_PLC  "LT-7130 LOLO ALARM SP PLC -> DeltaV"
  F23:185  LT_7130_HH_SP_PLC  "LT-7130 HIHI ALARM SP PLC -> DeltaV"
  F23:186  PDT_7110_LL_SP_PLC  "PDT-7110 LOLO ALARM SP PLC -> DeltaV"
  F23:187  PDT_7110_HH_SP_PLC  "PDT-7110 HIHI ALARM SP PLC -> DeltaV"
  F23:188  PT_7110_LL_SP_PLC  "PT-7110 LOLO ALARM SP PLC -> DeltaV"
  F23:189  PT_7110_HH_SP_PLC  "PT-7110 HIHI ALARM SP PLC -> DeltaV"
  F23:190  PT_7111_LL_SP_PLC  "PT-7111 LOLO ALARM SP PLC -> DeltaV"
  F23:191  PT_7111_HH_SP_PLC  "PT-7111 HIHI ALARM SP PLC -> DeltaV"
  F23:192  PT_7130_LL_SP_PLC  "PT-7130 LOLO ALARM SP PLC -> DeltaV"
  F23:193  PT_7130_HH_SP_PLC  "PT-7130 HIHI ALARM SP PLC -> DeltaV"
  F23:194  ST_7110_LL_SP_PLC  "ST-7110 LOLO ALARM SP PLC -> DeltaV"
  F23:195  ST_7110_HH_SP_PLC  "ST-7110 HIHI ALARM SP PLC -> DeltaV"
  F23:196  ST_7130_LL_SP_PLC  "ST-7130 LOLO ALARM SP PLC -> DeltaV"
  F23:197  ST_7130_HH_SP_PLC  "ST-7130 HIHI ALARM SP PLC -> DeltaV"
  F23:198  FT_7120_LL_SP_PLC  "FT-7120 LOLO ALARM SP PLC -> DeltaV"
  F23:199  FT_7120_HH_SP_PLC  "FT-7120 HIHI ALARM SP PLC -> DeltaV"
  F23:200  FT_7140_LL_SP_PLC  "FT-7140 LOLO ALARM SP PLC -> DeltaV"
  F23:201  FT_7140_HH_SP_PLC  "FT-7140 HIHI ALARM SP PLC -> DeltaV"
  F23:202  TT_7009_LL_SP_PLC  "TT-7009 LOLO ALARM SP PLC -> DeltaV"
  F23:203  TT_7009_HH_SP_PLC  "TT-7009 HIHI ALARM SP PLC -> DeltaV"
  F23:204  TT_7010_LL_SP_PLC  "TT-7010 LOLO ALARM SP PLC -> DeltaV"
  F23:205  TT_7010_HH_SP_PLC  "TT-7010 HIHI ALARM SP PLC -> DeltaV"
  F23:206  TT_7020_LL_SP_PLC  "TT-7020 LOLO ALARM SP PLC -> DeltaV"
  F23:207  TT_7020_HH_SP_PLC  "TT-7020 HIHI ALARM SP PLC -> DeltaV"
  F23:208  TT_7000_LL_SP_PLC  "TT-7000 LOLO ALARM SP PLC -> DeltaV"
  F23:209  TT_7000_HH_SP_PLC  "TT-7000 HIHI ALARM SP PLC -> DeltaV"
  F23:210  TT_7015_LL_SP_PLC  "TT-7015 LOLO ALARM SP PLC -> DeltaV"
  F23:211  TT_7015_HH_SP_PLC  "TT-7015 HIHI ALARM SP PLC -> DeltaV"
  F23:212  TT_7025_LL_SP_PLC  "TT-7025 LOLO ALARM SP PLC -> DeltaV"
  F23:213  TT_7025_HH_SP_PLC  "TT-7025 HIHI ALARM SP PLC -> DeltaV"
  F23:214  TT_7026_LL_SP_PLC  "TT-7026 LOLO ALARM SP PLC -> DeltaV"
  F23:215  TT_7026_HH_SP_PLC  "TT-7026 HIHI ALARM SP PLC -> DeltaV"
  F23:216  TT_7050_LL_SP_PLC  "TT-7050 LOLO ALARM SP PLC -> DeltaV"
  F23:217  TT_7050_HH_SP_PLC  "TT-7050 HIHI ALARM SP PLC -> DeltaV"
  F23:218  TT_7030_LL_SP_PLC  "TT-7030 LOLO ALARM SP PLC -> DeltaV"
  F23:219  TT_7030_HH_SP_PLC  "TT-7030 HIHI ALARM SP PLC -> DeltaV"
  F23:220  TT_7040_LL_SP_PLC  "TT-7040 LOLO ALARM SP PLC -> DeltaV"
  F23:221  TT_7040_HH_SP_PLC  "TT-7040 HIHI ALARM SP PLC -> DeltaV"
  F23:222  TT_7042_LL_SP_PLC  "TT-7042 LOLO ALARM SP PLC -> DeltaV"
  F23:223  TT_7042_HH_SP_PLC  "TT-7042 HIHI ALARM SP PLC -> DeltaV"
  F23:224  TT_7043_LL_SP_PLC  "TT-7043L LOLO ALARM SP PLC -> DeltaV"
  F23:225  TT_7043_HH_SP_PLC  "TT-7043L HIHI ALARM SP PLC -> DeltaV"
  F23:226  TT_7044_LL_SP_PLC  "TT-7043R LOLO ALARM SP PLC -> DeltaV"
  F23:227  TT_7044_HH_SP_PLC  "TT-7043R HIHI ALARM SP PLC -> DeltaV"
  F23:228  TT_7045_LL_SP_PLC  "TT-7045 LOLO ALARM SP PLC -> DeltaV"
  F23:229  TT_7045_HH_SP_PLC  "TT-7045 HIHI ALARM SP PLC -> DeltaV"
  F23:230  TT_7046_LL_SP_PLC  "TT-7046 LOLO ALARM SP PLC -> DeltaV"
  F23:231  TT_7046_HH_SP_PLC  "TT-7046 HIHI ALARM SP PLC -> DeltaV"
  F23:232  TT_7047_LL_SP_PLC  "TT-7047 LOLO ALARM SP PLC -> DeltaV"
  F23:233  TT_7047_HH_SP_PLC  "TT-7047 HIHI ALARM SP PLC -> DeltaV"
  F23:234  TT_7110_LL_SP_PLC  "TT-7110 LOLO ALARM SP PLC -> DeltaV"
  F23:235  TT_7110_HH_SP_PLC  "TT-7110 HIHI ALARM SP PLC -> DeltaV"
  F23:236  TT_7111_LL_SP_PLC  "TT-7111 LOLO ALARM SP PLC -> DeltaV"
  F23:237  TT_7111_HH_SP_PLC  "TT-7111 HIHI ALARM SP PLC -> DeltaV"
  F23:238  TT_7118_LL_SP_PLC  "TT-7118 LOLO ALARM SP PLC -> DeltaV"
  F23:239  TT_7118_HH_SP_PLC  "TT-7118 HIHI ALARM SP PLC -> DeltaV"
  F23:240  TT_7119_LL_SP_PLC  "TT-7119 LOLO ALARM SP PLC -> DeltaV"
  F23:241  TT_7119_HH_SP_PLC  "TT-7119 HIHI ALARM SP PLC -> DeltaV"
  F23:242  TT_7130_LL_SP_PLC  "TT-7130 LOLO ALARM SP PLC -> DeltaV"
  F23:243  TT_7130_HH_SP_PLC  "TT-7130 HIHI ALARM SP PLC -> DeltaV"
  F23:244  ST_7010_H_AL_SP_PLC  "FT-7140 HI ALARM SP PLC -> DeltaV"
  F23:245  ST_7010_HH_SP_PLC  "ST-7010 HIHI ALARM SP PLC -> DeltaV"
  F23:246  TT_7135_LL_SP_PLC  "TT-7135 LOLO ALARM SP PLC -> DeltaV"
  F23:247  TT_7135_HH_SP_PLC  "TT-7135 HIHI ALARM SP PLC -> DeltaV"
  F23:248  TT_7140_LL_SP_PLC  "TT-7140 LOLO ALARM SP PLC -> DeltaV"
  F23:249  TT_7140_HH_SP_PLC  "TT-7140 HIHI ALARM SP PLC -> DeltaV"
  F23:250  TT_7145_LL_SP_PLC  "TT-7145 LOLO ALARM SP PLC -> DeltaV"
  F23:251  TT_7145_HH_SP_PLC  "TT-7145 HIHI ALARM SP PLC -> DeltaV"
  F23:252  PT_7026_HH_SP_PLC  "PT-7026 HIHI ALARM SP PLC -> DeltaV"
  F23:253  PT_7026_H_AL_SP_PLC  "PT-7026 HI ALARM SP PLC -> DeltaV"
  F23:254  PT_7026_L_AL_SP_PLC  "PT-7026 LO ALARM SP PLC -> DeltaV"
  F23:255  PT_7026_LL_SP_PLC  "PT-7026 LOLO ALARM SP PLC -> DeltaV"
  F24:0  TT_7027_HH_SP_PLC  "TT-7027 HIHI ALARM SP PLC -> DeltaV"
  F24:1  TT_7027_H_AL_SP_PLC  "TT-7027 HI ALARM SP PLC -> DeltaV"
  F24:2  TT_7027_L_AL_SP_PLC  "TT-7027 LO ALARM SP PLC -> DeltaV"
  F24:3  TT_7027_LL_SP_PLC  "TT-7027 LOLO ALARM SP PLC -> DeltaV"
  F24:4  FIC7015_KC_PLC  "FIC7015 Kc PLC -> DeltaV"
  F24:5  FIC7015_TI_PLC  "FIC7015 Ti PLC -> DeltaV"
  F24:6  FIC7015_TD_PLC  "FIC7015 Td PLC -> DeltaV"
  F24:7  TIC7010_KC_PLC  "TIC7010 Kc PLC -> DeltaV"
  F24:8  TIC7010_TI_PLC  "TIC7010 Ti PLC -> DeltaV"
  F24:9  TIC7010_TD_PLC  "TIC7010_Td PLC -> DeltaV"
  F24:10  FIC7000_KC_PLC  "FIC7000 Kc PLC -> DeltaV"
  F24:11  FIC7000_TI_PLC  "FIC7000 Ti PLC -> DeltaV"
  F24:12  FIC7000_TD_PLC  "FIC7000 Td PLC -> DeltaV"
  F24:13  FIC7005_KC_PLC  "FIC7005 Kc PLC -> DeltaV"
  F24:14  FIC7005_TI_PLC  "FIC7005 Ti PLC -> DeltaV"
  F24:15  FIC7005_TD_PLC  "FIC7005 Td PLC -> DeltaV"
  F24:16  FIC7008_KC_PLC  "FIC7008 Kc PLC -> DeltaV"
  F24:17  FIC7008_TI_PLC  "FIC7008 Ti PLC -> DeltaV"
  F24:18  FIC7008_TD_PLC  "FIC7008 Td PLC -> DeltaV"
  F24:19  FIC7010_KC_PLC  "FIC7010 Kc PLC -> DeltaV"
  F24:20  FIC7010_TI_PLC  "FIC7010 Ti PLC -> DeltaV"
  F24:21  FIC7010_TD_PLC  "FIC7010_Td PLC -> DeltaV"
  F24:22  LIC7050_KC_PLC  "LIC7050 Kc PLC -> DeltaV"
  F24:23  LIC7050_TI_PLC  "LIC7050 Ti PLC -> DeltaV"
  F24:24  LIC7050_TD_PLC  "LIC7050 Td PLC -> DeltaV"
  F24:25  TIC7026_KC_PLC  "TIC7026 Kc PLC -> DeltaV"
  F24:26  TIC7026_TI_PLC  "TIC7026 Ti PLC -> DeltaV"
  F24:27  TIC7026_TD_PLC  "TIC7026 Td PLC -> DeltaV"
  F24:28  FIC7030_KC_PLC  "FIC7030 Kc PLC -> DeltaV"
  F24:29  FIC7030_TI_PLC  "FIC7030 Ti PLC -> DeltaV"
  F24:30  FIC7030_TD_PLC  "FIC7030 Td PLC -> DeltaV"
  F24:31  FIC7040_KC_PLC  "FIC7040 Kc PLC -> DeltaV"
  F24:32  FIC7040_TI_PLC  "FIC7040 Ti PLC -> DeltaV"
  F24:33  FIC7040_TD_PLC  "FIC7040 Td PLC -> DeltaV"
  F24:34  LIC7030_KC_PLC  "LIC7030 Kc PLC -> DeltaV"
  F24:35  LIC7030_TI_PLC  "LIC7030 Ti PLC -> DeltaV"
  F24:36  LIC7030_TD_PLC  "LIC7030 Td PLC -> DeltaV"
  F24:37  PIC7050_KC_PLC  "PIC7050 Kc PLC -> DeltaV"
  F24:38  PIC7050_TI_PLC  "PIC7050 Ti PLC -> DeltaV"
  F24:39  PIC7050_TD_PLC  "PIC7050 Td PLC -> DeltaV"
  F24:40  TIC7047_KC_PLC  "TIC7047 Kc PLC -> DeltaV"
  F24:41  TIC7047_TI_PLC  "TIC7047 Ti PLC -> DeltaV"
  F24:42  TIC7047_TD_PLC  "TIC7047 Td PLC -> DeltaV"
  F24:43  TIC7045_KC_PLC  "TIC7045 Kc PLC -> DeltaV"
  F24:44  TIC7045_TI_PLC  "TIC7045 Ti PLC -> DeltaV"
  F24:45  TIC7045_TD_PLC  "TIC7045 Td PLC -> DeltaV"
  F24:46  FIC7110_KC_PLC  "FIC7110 Kc PLC -> DeltaV"
  F24:47  FIC7110_TI_PLC  "FIC7110 Ti PLC -> DeltaV"
  F24:48  FIC7110_TD_PLC  "FIC7110 Td PLC -> DeltaV"
  F24:49  LIC7110_KC_PLC  "LIC7110 Kc PLC -> DeltaV"
  F24:50  LIC7110_TI_PLC  "LIC7110 Ti PLC -> DeltaV"
  F24:51  LIC7110_TD_PLC  "LIC7110 Td PLC -> DeltaV"
  F24:52  LIC7130_KC_PLC  "LIC7130 Kc PLC -> DeltaV"
  F24:53  LIC7130_TI_PLC  "LIC7130 Ti PLC -> DeltaV"
  F24:54  LIC7130_TD_PLC  "LIC7130 Td PLC -> DeltaV"
  F24:55  PIC7130_KC_PLC  "PIC7130 Kc PLC -> DeltaV"
  F24:56  PIC7130_TI_PLC  "PIC7130 Ti PLC -> DeltaV"
  F24:57  PIC7130_TD_PLC  "PIC7130 Td PLC -> DeltaV"
  F24:58  TIC7110_KC_PLC  "TIC7110 Kc PLC -> DeltaV"
  F24:59  TIC7110_TI_PLC  "TIC7110 Ti PLC -> DeltaV"
  F24:60  TIC7110_TD_PLC  "TIC7110 Td PLC -> DeltaV"
  F24:61  FIC7140_KC_PLC  "FIC7140 Kc PLC -> DeltaV"
  F24:62  FIC7140_TI_PLC  "FIC7140 Ti PLC -> DeltaV"
  F24:63  FIC7140_TD_PLC  "FIC7140 Td PLC -> DeltaV"
  F24:64  TIC7010_SP_PLC  "TIC7010 SP PLC -> DeltaV"
  F24:65  FIC7015_SP_PLC  "FIC7015 SP PLC -> DeltaV"
  F24:66  FIC7015_OP_PLC  "FIC7015 OP PLC -> DeltaV"
  F24:67  TIC7010_OP_PLC  "TIC7010 OP PLC -> DeltaV"
  F24:68  FIC7000_SP_PLC  "FIC7000 SP PLC -> DeltaV"
  F24:69  FIC7000_OP_PLC  "FIC7000 OP PLC -> DeltaV"
  F24:70  FIC7005_SP_PLC  "FIC7005 SP PLC -> DeltaV"
  F24:71  FIC7005_OP_PLC  "FIC7005 OP PLC -> DeltaV"
  F24:72  FIC7008_SP_PLC  "FIC7008 SP PLC -> DeltaV"
  F24:73  FIC7008_OP_PLC  "FIC7008 OP PLC -> DeltaV"
  F24:74  FIC7010_SP_PLC  "FIC7010 SP PLC -> DeltaV"
  F24:75  FIC7010_OP_PLC  "FIC7010 OP PLC -> DeltaV"
  F24:76  LIC7050_SP_PLC  "LIC7050 SP PLC -> DeltaV"
  F24:77  LIC7050_OP_PLC  "LIC7050 OP PLC -> DeltaV"
  F24:78  TIC7026_SP_PLC  "TIC7026 SP PLC -> DeltaV"
  F24:79  TIC7026_OP_PLC  "TIC7026 OP PLC -> DeltaV"
  F24:80  FIC7030_SP_PLC  "FIC7030 SP PLC -> DeltaV"
  F24:81  FIC7030_OP_PLC  "FIC7030 OP PLC -> DeltaV"
  F24:82  FIC7040_SP_PLC  "FIC7040 SP PLC -> DeltaV"
  F24:83  FIC7040_OP_PLC  "FIC7040 OP PLC -> DeltaV"
  F24:84  LIC7030_OP_PLC  "LIC7030 OP PLC -> DeltaV"
  F24:85  PIC7050_OP_PLC  "PIC7050 OP PLC -> DeltaV"
  F24:86  TIC7047_SP_PLC  "TIC7047 SP PLC -> DeltaV"
  F24:87  TIC7047_OP_PLC  "TIC7047 OP PLC -> DeltaV"
  F24:88  TIC7045_SP_PLC  "TIC7045 SP PLC -> DeltaV"
  F24:89  TIC7045_OP_PLC  "TIC7045 OP PLC -> DeltaV"
  F24:90  FIC7110_SP_PLC  "FIC7110 SP PLC -> DeltaV"
  F24:91  FIC7110_OP_PLC  "FIC7110 OP PLC -> DeltaV"
  F24:92  LIC7110_SP_PLC  "LIC7110 SP PLC -> DeltaV"
  F24:93  LIC7110_OP_PLC  "LIC7110 OP PLC -> DeltaV"
  F24:94  LIC7130_SP_PLC  "LIC7130 SP PLC -> DeltaV"
  F24:95  LIC7130_OP_PLC  "LIC7130 OP PLC -> DeltaV"
  F24:96  PIC7130_SP_PLC  "PIC7130 SP PLC -> DeltaV"
  F24:97  PIC7130_OP_PLC  "PIC7130 OP PLC -> DeltaV"
  F24:98  TIC7110_SP_PLC  "TIC7110 SP PLC -> DeltaV"
  F24:99  TIC7110_OP_PLC  "TIC7110 OP PLC -> DeltaV"
  F24:100  FIC7140_SP_PLC  "FIC7140 SP PLC -> DeltaV"
  F24:101  FIC7140_OP_PLC  "FIC7140 OP PLC -> DeltaV"
  F24:102  FT7002_L_AL_D_SP_PLC  "FT-7002 LO ALM DELAY SP PLC -> DeltaV"
  F24:103  FT7002_H_AL_D_SP_PLC  "FT-7002 HI ALM DELAY SP PLC -> DeltaV"
  F24:104  FT7010_L_AL_D_SP_PLC  "FT-7010 LO ALM DELAY SP PLC -> DeltaV"
  F24:105  FT7010_H_AL_D_SP_PLC  "FT-7010 HI ALM DELAY SP PLC -> DeltaV"
  F24:106  LT7010_L_AL_D_SP_PLC  "LT-7010 LO ALM DELAY SP PLC -> DeltaV"
  F24:107  LT7010_H_AL_D_SP_PLC  "LT-7010 HI ALM DELAY SP PLC -> DeltaV"
  F24:108  PT7010_L_AL_D_SP_PLC  "PT-7010 LO ALM DELAY SP PLC -> DeltaV"
  F24:109  PT7010_H_AL_D_SP_PLC  "PT-7010 HI ALM DELAY SP PLC -> DeltaV"
  F24:110  PT7020_L_AL_D_SP_PLC  "PT-7020 LO ALM DELAY SP PLC -> DeltaV"
  F24:111  PT7020_H_AL_D_SP_PLC  "PT-7020 HI ALM DELAY SP PLC -> DeltaV"
  F24:112  FT7000_L_AL_D_SP_PLC  "FT-7000 LO ALM DELAY SP PLC -> DeltaV"
  F24:113  FT7000_H_AL_D_SP_PLC  "FT-7000 HI ALM DELAY SP PLC -> DeltaV"
  F24:114  FT7005_L_AL_D_SP_PLC  "FT-7005 LO ALM DELAY SP PLC -> DeltaV"
  F24:115  FT7005_H_AL_D_SP_PLC  "FT-7005 HI ALM DELAY SP PLC -> DeltaV"
  F24:116  FT7008_L_AL_D_SP_PLC  "FT-7008 LO ALM DELAY SP PLC -> DeltaV"
  F24:117  FT7008_H_AL_D_SP_PLC  "FT-7008 HI ALM DELAY SP PLC -> DeltaV"
  F24:118  FT7025_L_AL_D_SP_PLC  "FT-7025 LO ALM DELAY SP PLC -> DeltaV"
  F24:119  FT7025_H_AL_D_SP_PLC  "FT-7025 HI ALM DELAY SP PLC -> DeltaV"
  F24:120  FT7050_L_AL_D_SP_PLC  "FT-7050 LO ALM DELAY SP PLC -> DeltaV"
  F24:121  FT7050_H_AL_D_SP_PLC  "FT-7050 HI ALM DELAY SP PLC -> DeltaV"
  F24:122  LT7050_L_AL_D_SP_PLC  "LT-7050 LO ALM DELAY SP PLC -> DeltaV"
  F24:123  LT7050_H_AL_D_SP_PLC  "LT-7050 HI ALM DELAY SP PLC -> DeltaV"
  F24:124  PT7000_L_AL_D_SP_PLC  "PT-7000 LO ALM DELAY SP PLC -> DeltaV"
  F24:125  PT7000_H_AL_D_SP_PLC  "PT-7000 HI ALM DELAY SP PLC -> DeltaV"
  F24:126  PT7015_L_AL_D_SP_PLC  "PT-7015 LO ALM DELAY SP PLC -> DeltaV"
  F24:127  PT7015_H_AL_D_SP_PLC  "PT-7015 HI ALM DELAY SP PLC -> DeltaV"
  F24:128  PT7025_L_AL_D_SP_PLC  "PT-7025 LO ALM DELAY SP PLC -> DeltaV"
  F24:129  PT7025_H_AL_D_SP_PLC  "PT-7025 HI ALM DELAY SP PLC -> DeltaV"
  F24:130  FT7030_L_AL_D_SP_PLC  "FT-7030 LO ALM DELAY SP PLC -> DeltaV"
  F24:131  FT7030_H_AL_D_SP_PLC  "FT-7030 HI ALM DELAY SP PLC -> DeltaV"
  F24:132  FT7040_L_AL_D_SP_PLC  "FT-7040 LO ALM DELAY SP PLC -> DeltaV"
  F24:133  FT7040_H_AL_D_SP_PLC  "FT-7040 HI ALM DELAY SP PLC -> DeltaV"
  F24:134  FT7052_L_AL_D_SP_PLC  "FT-7052 LO ALM DELAY SP PLC -> DeltaV"
  F24:135  FT7052_H_AL_D_SP_PLC  "FT-7052 HI ALM DELAY SP PLC -> DeltaV"
  F24:136  LT7030_L_AL_D_SP_PLC  "LT-7030 LO ALM DELAY SP PLC -> DeltaV"
  F24:137  LT7030_H_AL_D_SP_PLC  "LT-7030 HI ALM DELAY SP PLC -> DeltaV"
  F24:138  PDT7040_L_AL_D_PLC  "PDT-7040 LO ALM DELAY SP PLC -> DeltaV"
  F24:139  PDT7040_H_AL_D_PLC  "PDT-7040 HI ALM DELAY SP PLC -> DeltaV"
  F24:140  PT7030_L_AL_D_SP_PLC  "PT-7030 LO ALM DELAY SP PLC -> DeltaV"
  F24:141  PT7030_H_AL_D_SP_PLC  "PT-7030 HI ALM DELAY SP PLC -> DeltaV"
  F24:142  PT7040_L_AL_D_SP_PLC  "PT-7040 LO ALM DELAY SP PLC -> DeltaV"
  F24:143  PT7040_H_AL_D_SP_PLC  "PT-7040 HI ALM DELAY SP PLC -> DeltaV"
  F24:144  PT7050_L_AL_D_SP_PLC  "PT-7050 LO ALM DELAY SP PLC -> DeltaV"
  F24:145  PT7050_H_AL_D_SP_PLC  "PT-7050 HI ALM DELAY SP PLC -> DeltaV"
  F24:146  ST7040_L_AL_D_SP_PLC  "ST-7040 LO ALM DELAY SP PLC -> DeltaV"
  F24:147  ST7040_H_AL_D_SP_PLC  "ST-7040 HI ALM DELAY SP PLC -> DeltaV"
  F24:148  FT7095_L_AL_D_SP_PLC  "FT-7095 LO ALM DELAY SP PLC -> DeltaV"
  F24:149  FT7095_H_AL_D_SP_PLC  "FT-7095 HI ALM DELAY SP PLC -> DeltaV"
  F24:150  FT7110_L_AL_D_SP_PLC  "FT-7110 LO ALM DELAY SP PLC -> DeltaV"
  F24:151  FT7110_H_AL_D_SP_PLC  "FT-7110 HI ALM DELAY SP PLC -> DeltaV"
  F24:152  FT7130_L_AL_D_SP_PLC  "FT-7130 LO ALM DELAY SP PLC -> DeltaV"
  F24:153  FT7130_H_AL_D_SP_PLC  "FT-7130 HI ALM DELAY SP PLC -> DeltaV"
  F24:154  FT7132_L_AL_D_SP_PLC  "FT-7132 LO ALM DELAY SP PLC -> DeltaV"
  F24:155  FT7132_H_AL_D_SP_PLC  "FT-7132 HI ALM DELAY SP PLC -> DeltaV"
  F24:156  FT7145_L_AL_D_SP_PLC  "FT-7145 LO ALM DELAY SP PLC -> DeltaV"
  F24:157  FT7145_H_AL_D_SP_PLC  "FT-7145 HI ALM DELAY SP PLC -> DeltaV"
  F24:158  LT7110_L_AL_D_SP_PLC  "LT-7110 LO ALM DELAY SP PLC -> DeltaV"
  F24:159  LT7110_H_AL_D_SP_PLC  "LT-7110 HI ALM DELAY SP PLC -> DeltaV"
  F24:160  LT7130_L_AL_D_SP_PLC  "LT-7130 LO ALM DELAY SP PLC -> DeltaV"
  F24:161  LT7130_H_AL_D_SP_PLC  "LT-7130 HI ALM DELAY SP PLC -> DeltaV"
  F24:162  PDT7110_L_AL_D_PLC  "PDT-7110 LO ALM DELAY SP PLC -> DeltaV"
  F24:163  PDT7110_H_AL_D_PLC  "PDT-7110 HI ALM DELAY SP PLC -> DeltaV"
  F24:164  PT7110_L_AL_D_SP_PLC  "PT-7110 LO ALM DELAY SP PLC -> DeltaV"
  F24:165  PT7110_H_AL_D_SP_PLC  "PT-7110 HI ALM DELAY SP PLC -> DeltaV"
  F24:166  PT7111_L_AL_D_SP_PLC  "PT-7111 LO ALM DELAY SP PLC -> DeltaV"
  F24:167  PT7111_H_AL_D_SP_PLC  "PT-7111 HI ALM DELAY SP PLC -> DeltaV"
  F24:168  PT7130_L_AL_D_SP_PLC  "PT-7130 LO ALM DELAY SP PLC -> DeltaV"
  F24:169  PT7130_H_AL_D_SP_PLC  "PT-7130 HI ALM DELAY SP PLC -> DeltaV"
  F24:170  ST7110_L_AL_D_SP_PLC  "ST-7110 LO ALM DELAY SP PLC -> DeltaV"
  F24:171  ST7110_H_AL_D_SP_PLC  "ST-7110 HI ALM DELAY SP PLC -> DeltaV"
  F24:172  ST7130_L_AL_D_SP_PLC  "ST-7130 LO ALM DELAY SP PLC -> DeltaV"
  F24:173  ST7130_H_AL_D_SP_PLC  "ST-7130 HI ALM DELAY SP PLC -> DeltaV"
  F24:174  FT7120_L_AL_D_SP_PLC  "FT-7120 LO ALM DELAY SP PLC -> DeltaV"
  F24:175  FT7120_H_AL_D_SP_PLC  "FT-7120 HI ALM DELAY SP PLC -> DeltaV"
  F24:176  FT7140_L_AL_D_SP_PLC  "FT-7140 LO ALM DELAY SP PLC -> DeltaV"
  F24:177  FT7140_H_AL_D_SP_PLC  "FT-7140 HI ALM DELAY SP PLC -> DeltaV"
  F24:178  TT7009_L_AL_D_SP_PLC  "TT-7009 LO ALM DELAY SP PLC -> DeltaV"
  F24:179  TT7009_H_AL_D_SP_PLC  "TT-7009 HI ALM DELAY SP PLC -> DeltaV"
  F24:180  TT7010_L_AL_D_SP_PLC  "TT-7010 LO ALM DELAY SP PLC -> DeltaV"
  F24:181  TT7010_H_AL_D_SP_PLC  "TT-7010 HI ALM DELAY SP PLC -> DeltaV"
  F24:182  TT7020_L_AL_D_SP_PLC  "TT-7020 LO ALM DELAY SP PLC -> DeltaV"
  F24:183  TT7020_H_AL_D_SP_PLC  "TT-7020 HI ALM DELAY SP PLC -> DeltaV"
  F24:184  TT7000_L_AL_D_SP_PLC  "TT-7000 LO ALM DELAY SP PLC -> DeltaV"
  F24:185  TT7000_H_AL_D_SP_PLC  "TT-7000 HI ALM DELAY SP PLC -> DeltaV"
  F24:186  TT7015_L_AL_D_SP_PLC  "TT-7015 LO ALM DELAY SP PLC -> DeltaV"
  F24:187  TT7015_H_AL_D_SP_PLC  "TT-7015 HI ALM DELAY SP PLC -> DeltaV"
  F24:188  TT7025_L_AL_D_SP_PLC  "TT-7025 LO ALM DELAY SP PLC -> DeltaV"
  F24:189  TT7025_H_AL_D_SP_PLC  "TT-7025 HI ALM DELAY SP PLC -> DeltaV"
  F24:190  TT7026_L_AL_D_SP_PLC  "TT-7026 LO ALM DELAY SP PLC -> DeltaV"
  F24:191  TT7026_H_AL_D_SP_PLC  "TT-7026 HI ALM DELAY SP PLC -> DeltaV"
  F24:192  TT7050_L_AL_D_SP_PLC  "TT-7050 LO ALM DELAY SP PLC -> DeltaV"
  F24:193  TT7050_H_AL_D_SP_PLC  "TT-7050 HI ALM DELAY SP PLC -> DeltaV"
  F24:194  TT7030_L_AL_D_SP_PLC  "TT-7030 LO ALM DELAY SP PLC -> DeltaV"
  F24:195  TT7030_H_AL_D_SP_PLC  "TT-7030 HI ALM DELAY SP PLC -> DeltaV"
  F24:196  TT7040_L_AL_D_SP_PLC  "TT-7040 LO ALM DELAY SP PLC -> DeltaV"
  F24:197  TT7040_H_AL_D_SP_PLC  "TT-7040 HI ALM DELAY SP PLC -> DeltaV"
  F24:198  TT7042_L_AL_D_SP_PLC  "TT-7042 LO ALM DELAY SP PLC -> DeltaV"
  F24:199  TT7042_H_AL_D_SP_PLC  "TT-7042 HI ALM DELAY SP PLC -> DeltaV"
  F24:200  TT7043_L_AL_D_SP_PLC  "TT-7043 LO ALM DELAY SP PLC -> DeltaV"
  F24:201  TT7043_H_AL_D_SP_PLC  "TT-7043 HI ALM DELAY SP PLC -> DeltaV"
  F24:202  TT7044_L_AL_D_SP_PLC  "TT-7044 LO ALM DELAY SP PLC -> DeltaV"
  F24:203  TT7044_H_AL_D_SP_PLC  "TT-7044 HI ALM DELAY SP PLC -> DeltaV"
  F24:204  TT7045_L_AL_D_SP_PLC  "TT-7045 LO ALM DELAY SP PLC -> DeltaV"
  F24:205  TT7045_H_AL_D_SP_PLC  "TT-7045 HI ALM DELAY SP PLC -> DeltaV"
  F24:206  TT7046_L_AL_D_SP_PLC  "TT-7046 LO ALM DELAY SP PLC -> DeltaV"
  F24:207  TT7046_H_AL_D_SP_PLC  "TT-7046 HI ALM DELAY SP PLC -> DeltaV"
  F24:208  TT7047_L_AL_D_SP_PLC  "TT-7047 LO ALM DELAY SP PLC -> DeltaV"
  F24:209  TT7047_H_AL_D_SP_PLC  "TT-7047 HI ALM DELAY SP PLC -> DeltaV"
  F24:210  TT7110_L_AL_D_SP_PLC  "TT-7110 LO ALM DELAY SP PLC -> DeltaV"
  F24:211  TT7110_H_AL_D_SP_PLC  "TT-7110 HI ALM DELAY SP PLC -> DeltaV"
  F24:212  TT7111_L_AL_D_SP_PLC  "TT-7111 LO ALM DELAY SP PLC -> DeltaV"
  F24:213  TT7111_H_AL_D_SP_PLC  "TT-7111 HI ALM DELAY SP PLC -> DeltaV"
  F24:214  TT7118_L_AL_D_SP_PLC  "TT-7118 LO ALM DELAY SP PLC -> DeltaV"
  F24:215  TT7118_H_AL_D_SP_PLC  "TT-7118 HI ALM DELAY SP PLC -> DeltaV"
  F24:216  TT7119_L_AL_D_SP_PLC  "TT-7119 LO ALM DELAY SP PLC -> DeltaV"
  F24:217  TT7119_H_AL_D_SP_PLC  "TT-7119 HI ALM DELAY SP PLC -> DeltaV"
  F24:218  TT7130_L_AL_D_SP_PLC  "TT-7130 LO ALM DELAY SP PLC -> DeltaV"
  F24:219  TT7130_H_AL_D_SP_PLC  "TT-7130 HI ALM DELAY SP PLC -> DeltaV"
  F24:220  ST7010_LL_D_SP_PLC  "ST-7010 LL ALM DELAY SP PLC -> DeltaV"
  F24:221  ST7010_HH_D_SP_PLC  "ST-7010 HH ALM DELAY SP PLC -> DeltaV"
  F24:222  TT7135_L_AL_D_SP_PLC  "TT-7135 LO ALM DELAY SP PLC -> DeltaV"
  F24:223  TT7135_H_AL_D_SP_PLC  "TT-7135 HI ALM DELAY SP PLC -> DeltaV"
  F24:224  TT7140_L_AL_D_SP_PLC  "TT-7140 LO ALM DELAY SP PLC -> DeltaV"
  F24:225  TT7140_H_AL_D_SP_PLC  "TT-7140 HI ALM DELAY SP PLC -> DeltaV"
  F24:226  TT7145_L_AL_D_SP_PLC  "TT-7145 LO ALM DELAY SP PLC -> DeltaV"
  F24:227  TT7145_H_AL_D_SP_PLC  "TT-7145 HI ALM DELAY SP PLC -> DeltaV"
  F24:228  FT7002_LL_D_SP_PLC  "FT-7002 LOLO ALM DELAY SP PLC -> DeltaV"
  F24:229  FT7002_HH_D_SP_PLC  "FT-7002 HIHI ALM DELAY SP PLC -> DeltaV"
  F24:230  FT7010_LL_D_SP_PLC  "FT-7010 LOLO ALM DELAY SP PLC -> DeltaV"
  F24:231  FT7010_HH_D_SP_PLC  "FT-7010 HIHI ALM DELAY SP PLC -> DeltaV"
  F24:232  LT7010_LL_D_SP_PLC  "LT-7010 LOLO ALM DELAY SP PLC -> DeltaV"
  F24:233  LT7010_HH_D_SP_PLC  "LT-7010 HIHI ALM DELAY SP PLC -> DeltaV"
  F24:234  PT7010_LL_D_SP_PLC  "PT-7010 LOLO ALM DELAY SP PLC -> DeltaV"
  F24:235  PT7010_HH_D_SP_PLC  "PT-7010 HIHI ALM DELAY SP PLC -> DeltaV"
  F24:236  PT7020_LL_D_SP_PLC  "PT-7020 LOLO ALM DELAY SP PLC -> DeltaV"
  F24:237  PT7020_HH_D_SP_PLC  "PT-7020 HIHI ALM DELAY SP PLC -> DeltaV"
  F24:238  FT7000_LL_D_SP_PLC  "FT-7000 LOLO ALM DELAY SP PLC -> DeltaV"
  F24:239  FT7000_HH_D_SP_PLC  "FT-7000 HIHI ALM DELAY SP PLC -> DeltaV"
  F24:240  FT7005_LL_D_SP_PLC  "FT-7005 LOLO ALM DELAY SP PLC -> DeltaV"
  F24:241  FT7005_HH_D_SP_PLC  "FT-7005 HIHI ALM DELAY SP PLC -> DeltaV"
  F24:242  FT7008_LL_D_SP_PLC  "FT-7008 LOLO ALM DELAY SP PLC -> DeltaV"
  F24:243  FT7008_HH_D_SP_PLC  "FT-7008 HIHI ALM DELAY SP PLC -> DeltaV"
  F24:244  FT7025_LL_D_SP_PLC  "FT-7025 LOLO ALM DELAY SP PLC -> DeltaV"
  F24:245  FT7025_HH_D_SP_PLC  "FT-7025 HIHI ALM DELAY SP PLC -> DeltaV"
  F24:246  FT7050_LL_D_SP_PLC  "FT-7050 LOLO ALM DELAY SP PLC -> DeltaV"
  F24:247  FT7050_HH_D_SP_PLC  "FT-7050 HIHI ALM DELAY SP PLC -> DeltaV"
  F24:248  LT7050_LL_D_SP_PLC  "LT-7050 LOLO ALM DELAY SP PLC -> DeltaV"
  F24:249  LT7050_HH_D_SP_PLC  "LT-7050 HIHI ALM DELAY SP PLC -> DeltaV"
  F24:250  PT7000_LL_D_SP_PLC  "PT-7000 LOLO ALM DELAY SP PLC -> DeltaV"
  F24:251  PT7000_HH_D_SP_PLC  "PT-7000 HIHI ALM DELAY SP PLC -> DeltaV"
  F24:252  PT7015_LL_D_SP_PLC  "PT-7015 LOLO ALM DELAY SP PLC -> DeltaV"
  F24:253  PT7015_HH_D_SP_PLC  "PT-7015 HIHI ALM DELAY SP PLC -> DeltaV"
  F24:254  PT7025_LL_D_SP_PLC  "PT-7025 LOLO ALM DELAY SP PLC -> DeltaV"
  F24:255  PT7025_HH_D_SP_PLC  "PT-7025 HIHI ALM DELAY SP PLC -> DeltaV"
  F25:0  FT7030_LL_D_SP_PLC  "FT-7030 LOLO ALM DELAY SP PLC -> DeltaV"
  F25:1  FT7030_HH_D_SP_PLC  "FT-7030 HIHI ALM DELAY SP PLC -> DeltaV"
  F25:2  FT7040_LL_D_SP_PLC  "FT-7040 LOLO ALM DELAY SP PLC -> DeltaV"
  F25:3  FT7040_HH_D_SP_PLC  "FT-7040 HIHI ALM DELAY SP PLC -> DeltaV"
  F25:4  FT7052_LL_D_SP_PLC  "FT-7052 LOLO ALM DELAY SP PLC -> DeltaV"
  F25:5  FT7052_HH_D_SP_PLC  "FT-7052 HIHI ALM DELAY SP PLC -> DeltaV"
  F25:6  LT7030_LL_D_SP_PLC  "LT-7030 LOLO ALM DELAY SP PLC -> DeltaV"
  F25:7  LT7030_HH_D_SP_PLC  "LT-7030 HIHI ALM DELAY SP PLC -> DeltaV"
  F25:8  PDT7040_LL_D_SP_PLC  "PDT-7040 LOLO ALM DELAY SP PLC -> DeltaV"
  F25:9  PDT7040_HH_D_SP_PLC  "PDT-7040 HIHI ALM DELAY SP PLC -> DeltaV"
  F25:10  PT7030_LL_D_SP_PLC  "PT-7030 LOLO ALM DELAY SP PLC -> DeltaV"
  F25:11  PT7030_HH_D_SP_PLC  "PT-7030 HIHI ALM DELAY SP PLC -> DeltaV"
  F25:12  PT7040_LL_D_SP_PLC  "PT-7040 LOLO ALM DELAY SP PLC -> DeltaV"
  F25:13  PT7040_HH_D_SP_PLC  "PT-7040 HIHI ALM DELAY SP PLC -> DeltaV"
  F25:14  PT7050_LL_D_SP_PLC  "PT-7050 LOLO ALM DELAY SP PLC -> DeltaV"
  F25:15  PT7050_HH_D_SP_PLC  "PT-7050 HIHI ALM DELAY SP PLC -> DeltaV"
  F25:16  ST7040_LL_D_SP_PLC  "ST-7040 LOLO ALM DELAY SP PLC -> DeltaV"
  F25:17  ST7040_HH_D_SP_PLC  "ST-7040 HIHI ALM DELAY SP PLC -> DeltaV"
  F25:18  FT7095_LL_D_SP_PLC  "FT-7095 LOLO ALM DELAY SP PLC -> DeltaV"
  F25:19  FT7095_HH_D_SP_PLC  "FT-7095 HIHI ALM DELAY SP PLC -> DeltaV"
  F25:20  FT7110_LL_D_SP_PLC  "FT-7110 LOLO ALM DELAY SP PLC -> DeltaV"
  F25:21  FT7110_HH_D_SP_PLC  "FT-7110 HIHI ALM DELAY SP PLC -> DeltaV"
  F25:22  FT7130_LL_D_SP_PLC  "FT-7130 LOLO ALM DELAY SP PLC -> DeltaV"
  F25:23  FT7130_HH_D_SP_PLC  "FT-7130 HIHI ALM DELAY SP PLC -> DeltaV"
  F25:24  FT7132_LL_D_SP_PLC  "FT-7132 LOLO ALM DELAY SP PLC -> DeltaV"
  F25:25  FT7132_HH_D_SP_PLC  "FT-7132 HIHI ALM DELAY SP PLC -> DeltaV"
  F25:26  FT7145_LL_D_SP_PLC  "FT-7145 LOLO ALM DELAY SP PLC -> DeltaV"
  F25:27  FT7145_HH_D_SP_PLC  "FT-7145 HIHI ALM DELAY SP PLC -> DeltaV"
  F25:28  LT7110_LL_D_SP_PLC  "LT-7110 LOLO ALM DELAY SP PLC -> DeltaV"
  F25:29  LT7110_HH_D_SP_PLC  "LT-7110 HIHI ALM DELAY SP PLC -> DeltaV"
  F25:30  LT7130_LL_D_SP_PLC  "LT-7130 LOLO ALM DELAY SP PLC -> DeltaV"
  F25:31  LT7130_HH_D_SP_PLC  "LT-7130 HIHI ALM DELAY SP PLC -> DeltaV"
  F25:32  PDT7110_LL_D_SP_PLC  "PDT-7110 LOLO ALM DELAY SP PLC -> DeltaV"
  F25:33  PDT7110_HH_D_SP_PLC  "PDT-7110 HIHI ALM DELAY SP PLC -> DeltaV"
  F25:34  PT7110_LL_D_SP_PLC  "PT-7110 LOLO ALM DELAY SP PLC -> DeltaV"
  F25:35  PT7110_HH_D_SP_PLC  "PT-7110 HIHI ALM DELAY SP PLC -> DeltaV"
  F25:36  PT7111_LL_D_SP_PLC  "PT-7111 LOLO ALM DELAY SP PLC -> DeltaV"
  F25:37  PT7111_HH_D_SP_PLC  "PT-7111 HIHI ALM DELAY SP PLC -> DeltaV"
  F25:38  PT7130_LL_D_SP_PLC  "PT-7130 LOLO ALM DELAY SP PLC -> DeltaV"
  F25:39  PT7130_HH_D_SP_PLC  "PT-7130 HIHI ALM DELAY SP PLC -> DeltaV"
  F25:40  ST7110_LL_D_SP_PLC  "ST-7110 LOLO ALM DELAY SP PLC -> DeltaV"
  F25:41  ST7110_HH_D_SP_PLC  "ST-7110 HIHI ALM DELAY SP PLC -> DeltaV"
  F25:42  ST7130_LL_D_SP_PLC  "ST-7130 LOLO ALM DELAY SP PLC -> DeltaV"
  F25:43  ST7130_HH_D_SP_PLC  "ST-7130 HIHI ALM DELAY SP PLC -> DeltaV"
  F25:44  FT7120_LL_D_SP_PLC  "FT-7120 LOLO ALM DELAY SP PLC -> DeltaV"
  F25:45  FT7120_HH_D_SP_PLC  "FT-7120 HIHI ALM DELAY SP PLC -> DeltaV"
  F25:46  FT7140_LL_D_SP_PLC  "FT-7140 LOLO ALM DELAY SP PLC -> DeltaV"
  F25:47  FT7140_HH_D_SP_PLC  "FT-7140 HIHI ALM DELAY SP PLC -> DeltaV"
  F25:48  TT7009_LL_D_SP_PLC  "TT-7009 LOLO ALM DELAY SP PLC -> DeltaV"
  F25:49  TT7009_HH_D_SP_PLC  "TT-7009 HIHI ALM DELAY SP PLC -> DeltaV"
  F25:50  TT7010_LL_D_SP_PLC  "TT-7010 LOLO ALM DELAY SP PLC -> DeltaV"
  F25:51  TT7010_HH_D_SP_PLC  "TT-7010 HIHI ALM DELAY SP PLC -> DeltaV"
  F25:52  TT7020_LL_D_SP_PLC  "TT-7020 LOLO ALM DELAY SP PLC -> DeltaV"
  F25:53  TT7020_HH_D_SP_PLC  "TT-7020 HIHI ALM DELAY SP PLC -> DeltaV"
  F25:54  TT7000_LL_D_SP_PLC  "TT-7000 LOLO ALM DELAY SP PLC -> DeltaV"
  F25:55  TT7000_HH_D_SP_PLC  "TT-7000 HIHI ALM DELAY SP PLC -> DeltaV"
  F25:56  TT7015_LL_D_SP_PLC  "TT-7015 LOLO ALM DELAY SP PLC -> DeltaV"
  F25:57  TT7015_HH_D_SP_PLC  "TT-7015 HIHI ALM DELAY SP PLC -> DeltaV"
  F25:58  TT7025_LL_D_SP_PLC  "TT-7025 LOLO ALM DELAY SP PLC -> DeltaV"
  F25:59  TT7025_HH_DLY_SP_PLC  "TT-7025 HIHI ALM DELAY SP PLC -> DeltaV"
  F25:60  TT7026_LL_D_SP_PLC  "TT-7026 LOLO ALM DELAY SP PLC -> DeltaV"
  F25:61  TT7026_HH_D_SP_PLC  "TT-7026 HIHI ALM DELAY SP PLC -> DeltaV"
  F25:62  TT7050_LL_D_SP_PLC  "TT-7050 LOLO ALM DELAY SP PLC -> DeltaV"
  F25:63  TT7050_HH_D_SP_PLC  "TT-7050 HIHI ALM DELAY SP PLC -> DeltaV"
  F25:64  TT7030_LL_D_SP_PLC  "TT-7030 LOLO ALM DELAY SP PLC -> DeltaV"
  F25:65  TT7030_HH_D_SP_PLC  "TT-7030 HIHI ALM DELAY SP PLC -> DeltaV"
  F25:66  TT7040_LL_D_SP_PLC  "TT-7040 LOLO ALM DELAY SP PLC -> DeltaV"
  F25:67  TT7040_HH_D_SP_PLC  "TT-7040 HIHI ALM DELAY SP PLC -> DeltaV"
  F25:68  TT7042_LL_D_SP_PLC  "TT-7042 LOLO ALM DELAY SP PLC -> DeltaV"
  F25:69  TT7042_HH_D_SP_PLC  "TT-7042 HIHI ALM DELAY SP PLC -> DeltaV"
  F25:70  TT7043_LL_D_SP_PLC  "TT-7043 LOLO ALM DELAY SP PLC -> DeltaV"
  F25:71  TT7043_HH_D_SP_PLC  "TT-7043 HIHI ALM DELAY SP PLC -> DeltaV"
  F25:72  TT7044_LL_D_SP_PLC  "TT-7044 LOLO ALM DELAY SP PLC -> DeltaV"
  F25:73  TT7044_HH_D_SP_PLC  "TT-7044 HIHI ALM DELAY SP PLC -> DeltaV"
  F25:74  TT7045_LL_D_SP_PLC  "TT-7045 LOLO ALM DELAY SP PLC -> DeltaV"
  F25:75  TT7045_HH_D_SP_PLC  "TT-7045 HIHI ALM DELAY SP PLC -> DeltaV"
  F25:76  TT7046_LL_D_SP_PLC  "TT-7046 LOLO ALM DELAY SP PLC -> DeltaV"
  F25:77  TT7046_HH_D_SP_PLC  "TT-7046 HIHI ALM DELAY SP PLC -> DeltaV"
  F25:78  TT7047_LL_D_SP_PLC  "TT-7047 LOLO ALM DELAY SP PLC -> DeltaV"
  F25:79  TT7047_HH_D_SP_PLC  "TT-7047 HIHI ALM DELAY SP PLC -> DeltaV"
  F25:80  TT7110_LL_D_SP_PLC  "TT-7110 LOLO ALM DELAY SP PLC -> DeltaV"
  F25:81  TT7110_HH_D_SP_PLC  "TT-7110 HIHI ALM DELAY SP PLC -> DeltaV"
  F25:82  TT7111_LL_D_SP_PLC  "TT-7111 LOLO ALM DELAY SP PLC -> DeltaV"
  F25:83  TT7111_HH_D_SP_PLC  "TT-7111 HIHI ALM DELAY SP PLC -> DeltaV"
  F25:84  TT7118_LL_D_SP_PLC  "TT-7118 LOLO ALM DELAY SP PLC -> DeltaV"
  F25:85  TT7118_HH_D_SP_PLC  "TT-7118 HIHI ALM DELAY SP PLC -> DeltaV"
  F25:86  TT7119_LL_D_SP_PLC  "TT-7119 LOLO ALM DELAY SP PLC -> DeltaV"
  F25:87  TT7119_HH_D_SP_PLC  "TT-7119 HIHI ALM DELAY SP PLC -> DeltaV"
  F25:88  TT7130_LL_D_SP_PLC  "TT-7130 LOLO ALM DELAY SP PLC -> DeltaV"
  F25:89  TT7130_HH_D_SP_PLC  "TT-7130 HIHI ALM DELAY SP PLC -> DeltaV"
  F25:90  PT7026_LL_D_SP_PLC  "PT-7026 LL ALM DELAY SP PLC -> DeltaV"
  F25:91  PT7026_HH_D_SP_PLC  "PT-7026 HH ALM DELAY SP PLC -> DeltaV"
  F25:92  TT7135_LL_D_SP_PLC  "TT-7135 LOLO ALM DELAY SP PLC -> DeltaV"
  F25:93  TT7135_HH_D_SP_PLC  "TT-7135 HIHI ALM DELAY SP PLC -> DeltaV"
  F25:94  TT7140_LL_D_SP_PLC  "TT-7140 LOLO ALM DELAY SP PLC -> DeltaV"
  F25:95  TT7140_HH_D_SP_PLC  "TT-7140 HIHI ALM DELAY SP PLC -> DeltaV"
  F25:96  TT7145_LL_D_SP_PLC  "TT-7145 LOLO ALM DELAY SP PLC -> DeltaV"
  F25:97  TT7145_HH_D_SP_PLC  "TT-7145 HIHI ALM DELAY SP PLC -> DeltaV"
  F25:98  ST7010_L_AL_D_SP_PLC  "ST-7010 LO ALM DELAY SP PLC -> DeltaV"
  F25:99  ST7010_H_AL_D_SP_PLC  "ST-7010 HI ALM DELAY SP PLC -> DeltaV"
  F25:100  PT7026_L_AL_D_SP_PLC  "PT-7026 LO ALM DELAY SP PLC -> DeltaV"
  F25:101  PT7026_H_AL_D_SP_PLC  "PT-7026 HI ALM DELAY SP PLC -> DeltaV"
  F25:102  FIC7015_AUTO_MAN_PLC  "FIC7015 FT-7010 -> SY-7015 PLC -> DeltaV"
  F25:103  FIC7015_SP_MAX_PLC  "FIC7015 SY-7015 SP MAX (0-32767) PLC -> DeltaV"
  F25:104  FIC7015_SP_MIN_PLC  "FIC7015 SY-7015 SP MIN (0-32767) PLC -> DeltaV"
  F25:105  FIC7015_DB_PLC  "FIC7015 DB PLC -> DeltaV"
  F25:106  FIC7015_OP_MAX_PLC  "FIC7015 SY-7015 OP MAX (0-100%) PLC -> DeltaV"
  F25:107  FIC7015_OP_MIN_PLC  "FIC7015 SY-7015 OP MIN (0-100%) PLC -> DeltaV"
  F25:108  FIC7015_MAN_OP_PLC  "FIC7015 SY-7015 MAN OP (0-100%) PLC -> DeltaV"
  F25:109  TIC7010_AUTO_MAN_PLC  "TIC7010 TT-7010 -> TY-7010 PLC -> DeltaV"
  F25:110  TIC7010_SP_MAX_PLC  "TIC7010 TY-7010 SP MAX (0-32767) PLC -> DeltaV"
  F25:111  TIC7010_SP_MIN_PLC  "TIC7010 TY-7010 SP MIN (0-32767) PLC -> DeltaV"
  F25:112  TIC7010_DB_PLC  "TIC7010 DB PLC -> DeltaV"
  F25:113  TIC7010_OP_MAX_PLC  "TIC7010 TY-7010 OP MAX (0-100%) PLC -> DeltaV"
  F25:114  TIC7010_OP_MIN_PLC  "TIC7010 TY-7010 OP MIN (0-100%) PLC -> DeltaV"
  F25:115  TIC7010_MAN_OP_PLC  "TIC7010 TY-7010 MAN OP (0-100%) PLC -> DeltaV"
  F25:116  FIC7000_AUTO_MAN_PLC  "FIC7000 PT-7026 -> FY-7000 PLC -> DeltaV"
  F25:117  FIC7000_SP_MAX_PLC  "FIC7000 FY-7000 SP MAX (0-32767) PLC -> DeltaV"
  F25:118  FIC7000_SP_MIN_PLC  "FIC7000 FY-7000 SP MIN (0-32767) PLC -> DeltaV"
  F25:119  FIC7000_DB_PLC  "FIC7000 DB PLC -> DeltaV"
  F25:120  FIC7000_OP_MAX_PLC  "FIC7000 FY-7000 OP MAX (0-100%) PLC -> DeltaV"
  F25:121  FIC7000_OP_MIN_PLC  "FIC7000 FY-7000 OP MIN (0-100%) PLC -> DeltaV"
  F25:122  FIC7000_MAN_OP_PLC  "FIC7000 FY-7000 MAN OP (0-100%) PLC -> DeltaV"
  F25:123  FIC7005_AUTO_MAN_PLC  "FIC7005 FT-7005 -> FY-7005 PLC -> DeltaV"
  F25:124  FIC7005_SP_MAX_PLC  "FIC7005 FY-7005 SP MAX (0-32767) PLC -> DeltaV"
  F25:125  FIC7005_SP_MIN_PLC  "FIC7005 FY-7005 SP MIN (0-32767) PLC -> DeltaV"
  F25:126  FIC7005_DB_PLC  "FIC7005 DB PLC -> DeltaV"
  F25:127  FIC7005_OP_MAX_PLC  "FIC7005 FY-7005 OP MAX (0-100%) PLC -> DeltaV"
  F25:128  FIC7005_OP_MIN_PLC  "FIC7005 FY-7005 OP MIN (0-100%) PLC -> DeltaV"
  F25:129  FIC7005_MAN_OP_PLC  "FIC7005 FY-7005 MAN OP (0-100%) PLC -> DeltaV"
  F25:130  FIC7008_AUTO_MAN_PLC  "FIC7008 FT-7008 -> FY-7008 PLC -> DeltaV"
  F25:131  FIC7008_SP_MAX_PLC  "FIC7008 FY-7008 SP MAX (0-32767) PLC -> DeltaV"
  F25:132  FIC7008_SP_MIN_PLC  "FIC7008 FY-7008 SP MIN (0-32767) PLC -> DeltaV"
  F25:133  FIC7008_DB_PLC  "FIC7008 DB PLC -> DeltaV"
  F25:134  FIC7008_OP_MAX_PLC  "FIC7008 FY-7008 OP MAX (0-100%) PLC -> DeltaV"
  F25:135  FIC7008_OP_MIN_PLC  "FIC7008 FY-7008 OP MIN (0-100%) PLC -> DeltaV"
  F25:136  FIC7008_MAN_OP_PLC  "FIC7008 FY-7008 MAN OP (0-100%) PLC -> DeltaV"
  F25:137  FIC7010_AUTO_MAN_PLC  "FIC7010 FT-7010 -> FY-7010 PLC -> DeltaV"
  F25:138  FIC7010_SP_MAX_PLC  "FIC7010 FY-7010 SP MAX (0-32767) PLC -> DeltaV"
  F25:139  FIC7010_SP_MIN_PLC  "FIC7010 FY-7010 SP MIN (0-32767) PLC -> DeltaV"
  F25:140  FIC7010_DB_PLC  "FIC7010 DB PLC -> DeltaV"
  F25:141  FIC7010_OP_MAX_PLC  "FIC7010 FY-7010 OP MAX (0-100%) PLC -> DeltaV"
  F25:142  FIC7010_OP_MIN_PLC  "FIC7010 FY-7010 OP MIN (0-100%) PLC -> DeltaV"
  F25:143  FIC7010_MAN_OP_PLC  "FIC7010 FY-7010 MAN OP (0-100%) PLC -> DeltaV"
  F25:144  LIC7050_AUTO_MAN_PLC  "LIC7050 LT-7050 -> SY-7050 PLC -> DeltaV"
  F25:145  LIC7050_SP_MAX_PLC  "LIC7050 SY-7050 SP MAX (0-32767) PLC -> DeltaV"
  F25:146  LIC7050_SP_MIN_PLC  "LIC7050 SY-7050 SP MIN (0-32767) PLC -> DeltaV"
  F25:147  LIC7050_DB_PLC  "LIC7050 DB PLC -> DeltaV"
  F25:148  LIC7050_OP_MAX_PLC  "LIC7050 SY-7050 OP MAX (0-100%) PLC -> DeltaV"
  F25:149  LIC7050_OP_MIN_PLC  "LIC7050 SY-7050 OP MIN (0-100%) PLC -> DeltaV"
  F25:150  LIC7050_MAN_OP_PLC  "LIC7050 SY-7050 MAN OP (0-100%) PLC -> DeltaV"
  F25:151  TIC7026_AUTO_MAN_PLC  "TIC7026 TT-7026 -> SSR-7026 PLC -> DeltaV"
  F25:152  TIC7026_SP_MAX_PLC  "TIC7026 SSR-7026 SP MAX (0-32767) PLC -> DeltaV"
  F25:153  TIC7026_SP_MIN_PLC  "TIC7026 SSR-7026 SP MIN (0-32767) PLC -> DeltaV"
  F25:154  TIC7026_DB_PLC  "TIC7026 DB PLC -> DeltaV"
  F25:155  TIC7026_OP_MAX_PLC  "TIC7026 SSR-7026 OP MAX (0-100%) PLC -> DeltaV"
  F25:156  TIC7026_OP_MIN_PLC  "TIC7026 SSR-7026 OP MIN (0-100%) PLC -> DeltaV"
  F25:157  TIC7026_MAN_OP_PLC  "TIC7026 SSR-7026 MAN OP (0-100%) PLC -> DeltaV"
  F25:158  FIC7030_AUTO_MAN_PLC  "FIC7030 FT-7030 -> FY-7030 PLC -> DeltaV"
  F25:159  FIC7030_SP_MAX_PLC  "FIC7030 FY-7030 SP MAX (0-32767) PLC -> DeltaV"
  F25:160  FIC7030_SP_MIN_PLC  "FIC7030 FY-7030 SP MIN (0-32767) PLC -> DeltaV"
  F25:161  FIC7030_DB_PLC  "FIC7030 DB PLC -> DeltaV"
  F25:162  FIC7030_OP_MAX_PLC  "FIC7030 FY-7030 OP MAX (0-100%) PLC -> DeltaV"
  F25:163  FIC7030_OP_MIN_PLC  "FIC7030 FY-7030 OP MIN (0-100%) PLC -> DeltaV"
  F25:164  FIC7030_MAN_OP_PLC  "FIC7030 FY-7030 MAN OP (0-100%) PLC -> DeltaV"
  F25:165  FIC7040_AUTO_MAN_PLC  "FIC7040 FT-7040 -> FY-7040 PLC -> DeltaV"
  F25:166  FIC7040_SP_MAX_PLC  "FIC7040 FY-7040 SP MAX (0-32767) PLC -> DeltaV"
  F25:167  FIC7040_SP_MIN_PLC  "FIC7040 FY-7040 SP MIN (0-32767) PLC -> DeltaV"
  F25:168  FIC7040_DB_PLC  "FIC7040 DB PLC -> DeltaV"
  F25:169  FIC7040_OP_MAX_PLC  "FIC7040 FY-7040 OP MAX (0-100%) PLC -> DeltaV"
  F25:170  FIC7040_OP_MIN_PLC  "FIC7040 FY-7040 OP MIN (0-100%) PLC -> DeltaV"
  F25:171  FIC7040_MAN_OP_PLC  "FIC7040 FY-7040 MAN OP (0-100%) PLC -> DeltaV"
  F25:172  LIC7030_AUTO_MAN_PLC  "LIC7030 LT-7030 -> LY-7030 PLC -> DeltaV"
  F25:173  LIC7030_SP_MAX_PLC  "LIC7030 LY-7030 SP MAX (0-32767) PLC -> DeltaV"
  F25:174  LIC7030_SP_MIN_PLC  "LIC7030 LY-7030 SP MIN (0-32767) PLC -> DeltaV"
  F25:175  LIC7030_DB_PLC  "LIC7030 DB PLC -> DeltaV"
  F25:176  LIC7030_OP_MAX_PLC  "LIC7030 LY-7030 OP MAX (0-100%) PLC -> DeltaV"
  F25:177  LIC7030_OP_MIN_PLC  "LIC7030 LY-7030 OP MIN (0-100%) PLC -> DeltaV"
  F25:178  LIC7030_MAN_OP_PLC  "LIC7030 LY-7030 MAN OP (0-100%) PLC -> DeltaV"
  F25:179  PIC7050_AUTO_MAN_PLC  "PIC7050 PT-7050 -> PY-7050 PLC -> DeltaV"
  F25:180  PIC7050_SP_MAX_PLC  "PIC7050 PY-7050 SP MAX (0-32767) PLC -> DeltaV"
  F25:181  PIC7050_SP_MIN_PLC  "PIC7050 PY-7050 SP MIN (0-32767) PLC -> DeltaV"
  F25:182  PIC7050_DB_PLC  "PIC7050 DB PLC -> DeltaV"
  F25:183  PIC7050_OP_MAX_PLC  "PIC7050 PY-7050 OP MAX (0-100%) PLC -> DeltaV"
  F25:184  PIC7050_OP_MIN_PLC  "PIC7050 PY-7050 OP MIN (0-100%) PLC -> DeltaV"
  F25:185  PIC7050_MAN_OP_PLC  "PIC7050 PY-7050 MAN OP (0-100%) PLC -> DeltaV"
  F25:186  TIC7047_AUTO_MAN_PLC  "TIC7047 TT-7047 -> SSR-7047 PLC -> DeltaV"
  F25:187  TIC7047_SP_MAX_PLC  "TIC7047 SSR-7047 SP MAX (0-32767) PLC -> DeltaV"
  F25:188  TIC7047_SP_MIN_PLC  "TIC7047 SSR-7047 SP MIN (0-32767) PLC -> DeltaV"
  F25:189  TIC7047_DB_PLC  "TIC7047 DB PLC -> DeltaV"
  F25:190  TIC7047_OP_MAX_PLC  "TIC7047 SSR-7047 OP MAX (0-100%) PLC -> DeltaV"
  F25:191  TIC7047_OP_MIN_PLC  "TIC7047 SSR-7047 OP MIN (0-100%) PLC -> DeltaV"
  F25:192  TIC7047_MAN_OP_PLC  "TIC7047 SSR-7047 MAN OP (0-100%) PLC -> DeltaV"
  F25:193  TIC7045_AUTO_MAN_PLC  "TIC7045 TT-7045 -> TY-7045 PLC -> DeltaV"
  F25:194  TIC7045_SP_MAX_PLC  "TIC7045 TY-7045 SP MAX (0-32767) PLC -> DeltaV"
  F25:195  TIC7045_SP_MIN_PLC  "TIC7045 TY-7045 SP MIN (0-32767) PLC -> DeltaV"
  F25:196  TIC7045_DB_PLC  "TIC7045 DB PLC -> DeltaV"
  F25:197  TIC7045_OP_MAX_PLC  "TIC7045 TY-7045 OP MAX (0-100%) PLC -> DeltaV"
  F25:198  TIC7045_OP_MIN_PLC  "TIC7045 TY-7045 OP MIN (0-100%) PLC -> DeltaV"
  F25:199  TIC7045_MAN_OP_PLC  "TIC7045 TY-7045 MAN OP (0-100%) PLC -> DeltaV"
  F25:200  FIC7110_AUTO_MAN_PLC  "FIC7110 FT-7110 -> FY-7110 PLC -> DeltaV"
  F25:201  FIC7110_SP_MAX_PLC  "FIC7110 FY-7110 SP MAX (0-32767) PLC -> DeltaV"
  F25:202  FIC7110_SP_MIN_PLC  "FIC7110 FY-7110 SP MIN (0-32767) PLC -> DeltaV"
  F25:203  FIC7110_DB_PLC  "FIC7110 DB PLC -> DeltaV"
  F25:204  FIC7110_OP_MAX_PLC  "FIC7110 FY-7110 OP MAX (0-100%) PLC -> DeltaV"
  F25:205  FIC7110_OP_MIN_PLC  "FIC7110 FY-7110 OP MIN (0-100%) PLC -> DeltaV"
  F25:206  FIC7110_MAN_OP_PLC  "FIC7110 FY-7110 MAN OP (0-100%) PLC -> DeltaV"
  F25:207  LIC7110_AUTO_MAN_PLC  "LIC7110 LT-7110 -> LY-7110 PLC -> DeltaV"
  F25:208  LIC7110_SP_MAX_PLC  "LIC7110 LY-7110 SP MAX (0-32767) PLC -> DeltaV"
  F25:209  LIC7110_SP_MIN_PLC  "LIC7110 LY-7110 SP MIN (0-32767) PLC -> DeltaV"
  F25:210  LIC7110_DB_PLC  "LIC7110 DB PLC -> DeltaV"
  F25:211  LIC7110_OP_MAX_PLC  "LIC7110 LY-7110 OP MAX (0-100%) PLC -> DeltaV"
  F25:212  LIC7110_OP_MIN_PLC  "LIC7110 LY-7110 OP MIN (0-100%) PLC -> DeltaV"
  F25:213  LIC7110_MAN_OP_PLC  "LIC7110 LY-7110 MAN OP (0-100%) PLC -> DeltaV"
  F25:214  LIC7130_AUTO_MAN_PLC  "LIC7130 LT-7130 -> LY-7130 PLC -> DeltaV"
  F25:215  LIC7130_SP_MAX_PLC  "LIC7130 LY-7130 SP MAX (0-32767) PLC -> DeltaV"
  F25:216  LIC7130_SP_MIN_PLC  "LIC7130 LY-7130 SP MIN (0-32767) PLC -> DeltaV"
  F25:217  LIC7130_DB_PLC  "LIC7130 DB PLC -> DeltaV"
  F25:218  LIC7130_OP_MAX_PLC  "LIC7130 LY-7130 OP MAX (0-100%) PLC -> DeltaV"
  F25:219  LIC7130_OP_MIN_PLC  "LIC7130 LY-7130 OP MIN (0-100%) PLC -> DeltaV"
  F25:220  LIC7130_MAN_OP_PLC  "LIC7130 LY-7130 MAN OP (0-100%) PLC -> DeltaV"
  F25:221  PIC7130_AUTO_MAN_PLC  "PIC7130 PT-7130 -> PY-7130 PLC -> DeltaV"
  F25:222  PIC7130_SP_MAX_PLC  "PIC7130 PY-7130 SP MAX (0-32767) PLC -> DeltaV"
  F25:223  PIC7130_SP_MIN_PLC  "PIC7130 PY-7130 SP MIN (0-32767) PLC -> DeltaV"
  F25:224  PIC7130_DB_PLC  "PIC7130 DB PLC -> DeltaV"
  F25:225  PIC7130_OP_MAX_PLC  "PIC7130 PY-7130 OP MAX (0-100%) PLC -> DeltaV"
  F25:226  PIC7130_OP_MIN_PLC  "PIC7130 PY-7130 OP MIN (0-100%) PLC -> DeltaV"
  F25:227  PIC7130_MAN_OP_PLC  "PIC7130 PY-7130 MAN OP (0-100%) PLC -> DeltaV"
  F25:228  TIC7110_AUTO_MAN_PLC  "TIC7110 TT-7110 -> TY-7110 PLC -> DeltaV"
  F25:229  TIC7110_SP_MAX_PLC  "TIC7110 TY-7110 SP MAX (0-32767) PLC -> DeltaV"
  F25:230  TIC7110_SP_MIN_PLC  "TIC7110 TY-7110 SP MIN (0-32767) PLC -> DeltaV"
  F25:231  TIC7110_DB_PLC  "TIC7110 DB PLC -> DeltaV"
  F25:232  TIC7110_OP_MAX_PLC  "TIC7110 TY-7110 OP MAX (0-100%) PLC -> DeltaV"
  F25:233  TIC7110_OP_MIN_PLC  "TIC7110 TY-7110 OP MIN (0-100%) PLC -> DeltaV"
  F25:234  TIC7110_MAN_OP_PLC  "TIC7110 TY-7110 MAN OP (0-100%) PLC -> DeltaV"
  F25:235  FIC7140_AUTO_MAN_PLC  "FIC7140 FT-7140 -> FY-7140 PLC -> DeltaV"
  F25:236  FIC7140_SP_MAX_PLC  "FIC7140 FY-7140 SP MAX (0-32767) PLC -> DeltaV"
  F25:237  FIC7140_SP_MIN_PLC  "FIC7140 FY-7140 SP MIN (0-32767) PLC -> DeltaV"
  F25:238  FIC7140_DB_PLC  "FIC7140 DB PLC -> DeltaV"
  F25:239  FIC7140_OP_MAX_PLC  "FIC7140 FY-7140 OP MAX (0-100%) PLC -> DeltaV"
  F25:240  FIC7140_OP_MIN_PLC  "FIC7140 FY-7140 OP MIN (0-100%) PLC -> DeltaV"
  F25:241  FIC7140_MAN_OP_PLC  "FIC7140 FY-7140 MAN OP (0-100%) PLC -> DeltaV"
  F25:242  TT7027_LL_D_SP_PLC  "TT-7027 LOLO ALARM DELAY PLC -> DeltaV"
  F25:243  TT7027_HH_D_SP_PLC  "TT-7027 HIHI ALARM DELAY PLC -> DeltaV"
  F25:244  TT7027_L_AL_D_SP_PLC  "TT-7027 LO ALARM DELAY PLC -> DeltaV"
  F25:245  TT7027_H_AL_D_SP_PLC  "TT-7027 HI ALARM DELAY PLC -> DeltaV"
  F25:246  LSH_7131_DLY_SP_PLC  "LSH-7130 HIGH LEVEL ALARM DELAY PLC -> DeltaV"
  F25:247  LSH_7031_DLY_SP_PLC  "LSH-7031 HIGH LEVEL ALARM DELAY PLC -> DeltaV"
  F25:248  LIC7030_SP_DV  "LIC7030 SP DeltaV -> PLC"
  F25:249  PIC7050_SP_DV  "PIC7050 SP DeltaV -> PLC"
  F26:0  FT_7002_L_AL_SP_DV  "FT-7002 LO ALARM SP DeltaV -> PLC"
  F26:1  FT_7002_H_AL_SP_DV  "FT-7002 HI ALARM SP DeltaV -> PLC"
  F26:2  FT_7010_L_AL_SP_DV  "FT-7010 LO ALARM SP DeltaV -> PLC"
  F26:3  FT_7010_H_AL_SP_DV  "FT-7010 HI ALARM SP DeltaV -> PLC"
  F26:4  LT_7010_L_AL_SP_DV  "LT-7010 LO ALARM SP DeltaV -> PLC"
  F26:5  LT_7010_H_AL_SP_DV  "LT-7010 HI ALARM SP DeltaV -> PLC"
  F26:6  PT_7010_L_AL_SP_DV  "PT-7010 LO ALARM SP DeltaV -> PLC"
  F26:7  PT_7010_H_AL_SP_DV  "PT-7010 HI ALARM SP DeltaV -> PLC"
  F26:8  PT_7020_L_AL_SP_DV  "PT-7020 LO ALARM SP DeltaV -> PLC"
  F26:9  PT_7020_H_AL_SP_DV  "PT-7020 HI ALARM SP DeltaV -> PLC"
  F26:10  FT_7000_L_AL_SP_DV  "FT-7000 LO ALARM SP DeltaV -> PLC"
  F26:11  FT_7000_H_AL_SP_DV  "FT-7000 HI ALARM SP DeltaV -> PLC"
  F26:12  FT_7005_L_AL_SP_DV  "FT-7005 LO ALARM SP DeltaV -> PLC"
  F26:13  FT_7005_H_AL_SP_DV  "FT-7005 HI ALARM SP DeltaV -> PLC"
  F26:14  FT_7008_L_AL_SP_DV  "FT-7008 LO ALARM SP DeltaV -> PLC"
  F26:15  FT_7008_H_AL_SP_DV  "FT-7008 HI ALARM SP DeltaV -> PLC"
  F26:16  FT_7025_L_AL_SP_DV  "FT-7025 LO ALARM SP DeltaV -> PLC"
  F26:17  FT_7025_H_AL_SP_DV  "FT-7025 HI ALARM SP DeltaV -> PLC"
  F26:18  FT_7050_L_AL_SP_DV  "FT-7050 LO ALARM SP DeltaV -> PLC"
  F26:19  FT_7050_H_AL_SP_DV  "FT-7050 HI ALARM SP DeltaV -> PLC"
  F26:20  LT_7050_L_AL_SP_DV  "LT-7050 LO ALARM SP DeltaV -> PLC"
  F26:21  LT_7050_H_AL_SP_DV  "LT-7050 HI ALARM SP DeltaV -> PLC"
  F26:22  PT_7000_L_AL_SP_DV  "PT-7000 LO ALARM SP DeltaV -> PLC"
  F26:23  PT_7000_H_AL_SP_DV  "PT-7000 HI ALARM SP DeltaV -> PLC"
  F26:24  PT_7015_L_AL_SP_DV  "PT-7015 LO ALARM SP DeltaV -> PLC"
  F26:25  PT_7015_H_AL_SP_DV  "PT-7015 HI ALARM SP DeltaV -> PLC"
  F26:26  PT_7025_L_AL_SP_DV  "PT-7025 LO ALARM SP DeltaV -> PLC"
  F26:27  PT_7025_H_AL_SP_DV  "PT-7025 HI ALARM SP DeltaV -> PLC"
  F26:28  FT_7030_L_AL_SP_DV  "FT-7030 LO ALARM SP DeltaV -> PLC"
  F26:29  FT_7030_H_AL_SP_DV  "FT-7030 HI ALARM SP DeltaV -> PLC"
  F26:30  FT_7040_L_ALSP_DV  "FT-7040 LO ALARM SP DeltaV -> PLC"
  F26:31  FT_7040_H_AL_SP_DV  "FT-7040 HI ALARM SP DeltaV -> PLC"
  F26:32  FT_7052_L_AL_SP_DV  "FT-7052 LO ALARM SP DeltaV -> PLC"
  F26:33  FT_7052_H_AL_SP_DV  "FT-7052 HI ALARM SP DeltaV -> PLC"
  F26:34  LT_7030_L_AL_SP_DV  "LT-7030 LO ALARM SP DeltaV -> PLC"
  F26:35  LT_7030_H_AL_SP_DV  "LT-7030 HI ALARM SP DeltaV -> PLC"
  F26:36  PDT_7040_L_AL_SP_DV  "PDT-7040 LO ALARM SP DeltaV -> PLC"
  F26:37  PDT_7040_H_AL_SP_DV  "PDT-7040 HI ALARM SP DeltaV -> PLC"
  F26:38  PT_7030_L_AL_SP_DV  "PT-7030 LO ALARM SP DeltaV -> PLC"
  F26:39  PT_7030_H_AL_SP_DV  "PT-7030 HI ALARM SP DeltaV -> PLC"
  F26:40  PT_7040_L_AL_SP_DV  "PT-7040 LO ALARM SP DeltaV -> PLC"
  F26:41  PT_7040_H_AL_SP_DV  "PT-7040 HI ALARM SP DeltaV -> PLC"
  F26:42  PT_7050_L_AL_SP_DV  "PT-7050 LO ALARM SP DeltaV -> PLC"
  F26:43  PT_7050_H_AL_SP_DV  "PT-7050 HI ALARM SP DeltaV -> PLC"
  F26:44  ST_7040_L_AL_SP_DV  "ST-7040 LO ALARM SP DeltaV -> PLC"
  F26:45  ST_7040_H_AL_SP_DV  "ST-7040 HI ALARM SP DeltaV -> PLC"
  F26:46  FT_7095_L_AL_SP_DV  "FT-7095 LO ALARM SP DeltaV -> PLC"
  F26:47  FT_7095_H_AL_SP_DV  "FT-7095 HI ALARM SP DeltaV -> PLC"
  F26:48  FT_7110_L_AL_SP_DV  "FT-7110 LO ALARM SP DeltaV -> PLC"
  F26:49  FT_7110_H_AL_SP_DV  "FT-7110 HI ALARM SP DeltaV -> PLC"
  F26:50  FT_7130_L_AL_SP_DV  "FT-7130 LO ALARM SP DeltaV -> PLC"
  F26:51  FT_7130_H_AL_SP_DV  "FT-7130 HI ALARM SP DeltaV -> PLC"
  F26:52  FT_7132_L_AL_SP_DV  "FT-7132 LO ALARM SP DeltaV -> PLC"
  F26:53  FT_7132_H_AL_SP_DV  "FT-7132 HI ALARM SP DeltaV -> PLC"
  F26:54  FT_7145_L_AL_SP_DV  "FT-7145 LO ALARM SP DeltaV -> PLC"
  F26:55  FT_7145_H_AL_SP_DV  "FT-7145 HI ALARM SP DeltaV -> PLC"
  F26:56  LT_7110_L_AL_SP_DV  "LT-7110 LO ALARM SP DeltaV -> PLC"
  F26:57  LT_7110_H_AL_SP_DV  "LT-7110 HI ALARM SP DeltaV -> PLC"
  F26:58  LT_7130_L_AL_SP_DV  "LT-7130 LO ALARM SP DeltaV -> PLC"
  F26:59  LT_7130_H_AL_SP_DV  "LT-7130 HI ALARM SP DeltaV -> PLC"
  F26:60  PDT_7110_L_AL_SP_DV  "PDT-7110 LO ALARM SP DeltaV -> PLC"
  F26:61  PDT_7110_H_AL_SP_DV  "PDT-7110 HI ALARM SP DeltaV -> PLC"
  F26:62  PT_7110_L_AL_SP_DV  "PT-7110 LO ALARM SP DeltaV -> PLC"
  F26:63  PT_7110_H_AL_SP_DV  "PT-7110 HI ALARM SP DeltaV -> PLC"
  F26:64  PT_7111_L_AL_SP_DV  "PT-7111 LO ALARM SP DeltaV -> PLC"
  F26:65  PT_7111_H_AL_SP_DV  "PT-7111 HI ALARM SP DeltaV -> PLC"
  F26:66  PT_7130_L_AL_SP_DV  "PT-7130 LO ALARM SP DeltaV -> PLC"
  F26:67  PT_7130_H_AL_SP_DV  "PT-7130 HI ALARM SP DeltaV -> PLC"
  F26:68  ST_7110_L_AL_SP_DV  "ST-7110 LO ALARM SP DeltaV -> PLC"
  F26:69  ST_7110_H_AL_SP_DV  "ST-7110 HI ALARM SP DeltaV -> PLC"
  F26:70  ST_7130_L_AL_SP_DV  "ST-7130 LO ALARM SP DeltaV -> PLC"
  F26:71  ST_7130_H_AL_SP_DV  "ST-7130 HI ALARM SP DeltaV -> PLC"
  F26:72  FT_7120_L_AL_SP_DV  "FT-7120 LO ALARM SP DeltaV -> PLC"
  F26:73  FT_7120_H_AL_SP_DV  "FT-7120 HI ALARM SP DeltaV -> PLC"
  F26:74  FT_7140_L_AL_SP_DV  "FT-7140 LO ALARM SP DeltaV -> PLC"
  F26:75  FT_7140_H_AL_SP_DV  "FT-7140 HI ALARM SP DeltaV -> PLC"
  F26:76  TT_7009_L_AL_SP_DV  "TT-7009 LO ALARM SP DeltaV -> PLC"
  F26:77  TT_7009_H_AL_SP_DV  "TT-7009 HI ALARM SP DeltaV -> PLC"
  F26:78  TT_7010_L_AL_SP_DV  "TT-7010 LO ALARM SP DeltaV -> PLC"
  F26:79  TT_7010_H_AL_SP_DV  "TT-7010 HI ALARM SP DeltaV -> PLC"
  F26:80  TT_7020_L_AL_SP_DV  "TT-7020 LO ALARM SP DeltaV -> PLC"
  F26:81  TT_7020_H_AL_SP_DV  "TT-7020 HI ALARM SP DeltaV -> PLC"
  F26:82  TT_7000_L_AL_SP_DV  "TT-7000 LO ALARM SP DeltaV -> PLC"
  F26:83  TT_7000_H_AL_SP_DV  "TT-7000 HI ALARM SP DeltaV -> PLC"
  F26:84  TT_7015_L_AL_SP_DV  "TT-7015 LO ALARM SP DeltaV -> PLC"
  F26:85  TT_7015_H_AL_SP_DV  "TT-7015 HI ALARM SP DeltaV -> PLC"
  F26:86  TT_7025_L_AL_SP_DV  "TT-7025 LO ALARM SP DeltaV -> PLC"
  F26:87  TT_7025_H_AL_SP_DV  "TT-7025 HI ALARM SP DeltaV -> PLC"
  F26:88  TT_7026_L_AL_SP_DV  "TT-7026 LO ALARM SP DeltaV -> PLC"
  F26:89  TT_7026_H_AL_SP_DV  "TT-7026 HI ALARM SP DeltaV -> PLC"
  F26:90  TT_7050_L_AL_SP_DV  "TT-7050 LO ALARM SP DeltaV -> PLC"
  F26:91  TT_7050_H_AL_SP_DV  "TT-7050 HI ALARM SP DeltaV -> PLC"
  F26:92  TT_7030_L_AL_SP_DV  "TT-7030 LO ALARM SP DeltaV -> PLC"
  F26:93  TT_7030_H_AL_SP_DV  "TT-7030 HI ALARM SP DeltaV -> PLC"
  F26:94  TT_7040_L_AL_SP_DV  "TT-7040 LO ALARM SP DeltaV -> PLC"
  F26:95  TT_7040_H_AL_SP_DV  "TT-7040 HI ALARM SP DeltaV -> PLC"
  F26:96  TT_7042_L_AL_SP_DV  "TT-7042 LO ALARM SP DeltaV -> PLC"
  F26:97  TT_7042_H_AL_SP_DV  "TT-7042 HI ALARM SP DeltaV -> PLC"
  F26:98  TT_7043_L_AL_SP_DV  "TT-7043L LO ALARM SP DeltaV -> PLC"
  F26:99  TT_7043_H_AL_SP_DV  "TT-7043L HI ALARM SP DeltaV -> PLC"
  F26:100  TT_7044_L_AL_SP_DV  "TT-7043R LO ALARM SP DeltaV -> PLC"
  F26:101  TT_7044_H_AL_SP_DV  "TT-7043R HI ALARM SP DeltaV -> PLC"
  F26:102  TT_7045_L_AL_SP_DV  "TT-7045 LO ALARM SP DeltaV -> PLC"
  F26:103  TT_7045_H_AL_SP_DV  "TT-7045 HI ALARM SP DeltaV -> PLC"
  F26:104  TT_7046_L_AL_SP_DV  "TT-7046 LO ALARM SP DeltaV -> PLC"
  F26:105  TT_7046_H_AL_SP_DV  "TT-7046 HI ALARM SP DeltaV -> PLC"
  F26:106  TT_7047_L_AL_SP_DV  "TT-7047 LO ALARM SP DeltaV -> PLC"
  F26:107  TT_7047_H_AL_SP_DV  "TT-7047 HI ALARM SP DeltaV -> PLC"
  F26:108  TT_7110_L_AL_SP_DV  "TT-7110 LO ALARM SP DeltaV -> PLC"
  F26:109  TT_7110_H_AL_SP_DV  "TT-7110 HI ALARM SP DeltaV -> PLC"
  F26:110  TT_7111_L_AL_SP_DV  "TT-7111 LO ALARM SP DeltaV -> PLC"
  F26:111  TT_7111_H_AL_SP_DV  "TT-7111 HI ALARM SP DeltaV -> PLC"
  F26:112  TT_7118_L_AL_SP_DV  "TT-7118 LO ALARM SP DeltaV -> PLC"
  F26:113  TT_7118_H_AL_SP_DV  "TT-7118 HI ALARM SP DeltaV -> PLC"
  F26:114  TT_7119_L_AL_SP_DV  "TT-7119 LO ALARM SP DeltaV -> PLC"
  F26:115  TT_7119_H_AL_SP_DV  "TT-7119 HI ALARM SP DeltaV -> PLC"
  F26:116  TT_7130_L_AL_SP_DV  "TT-7130 LO ALARM SP DeltaV -> PLC"
  F26:117  TT_7130_H_AL_SP_DV  "TT-7130 HI ALARM SP DeltaV -> PLC"
  F26:118  ST_7010_LL_SP_DV  "ST-7010 LOLO ALARM SP DeltaV -> PLC"
  F26:119  ST_7010_L_AL_SP_DV  "ST-7010 LO ALARM SP DeltaV -> PLC"
  F26:120  TT_7135_L_AL_SP_DV  "TT-7135 LO ALARM SP DeltaV -> PLC"
  F26:121  TT_7135_H_AL_SP_DV  "TT-7135 HI ALARM SP DeltaV -> PLC"
  F26:122  TT_7140_L_AL_SP_DV  "TT-7140 LO ALARM SP DeltaV -> PLC"
  F26:123  TT_7140_H_AL_SP_DV  "TT-7140 HI ALARM SP DeltaV -> PLC"
  F26:124  TT_7145_L_AL_SP_DV  "TT-7145 LO ALARM SP DeltaV -> PLC"
  F26:125  TT_7145_H_AL_SP_DV  "TT-7145 HI ALARM SP DeltaV -> PLC"
  F26:126  FT_7002_LL_SP_DV  "FT-7002 LOLO ALARM SP DeltaV -> PLC"
  F26:127  FT_7002_HH_SP_DV  "FT-7002 HIHI ALARM SP DeltaV -> PLC"
  F26:128  FT_7010_LL_SP_DV  "FT-7010 LOLO ALARM SP DeltaV -> PLC"
  F26:129  FT_7010_HH_SP_DV  "FT-7010 HIHI ALARM SP DeltaV -> PLC"
  F26:130  LT_7010_LL_SP_DV  "LT-7010 LOLO ALARM SP DeltaV -> PLC"
  F26:131  LT_7010_HH_SP_DV  "LT-7010 HIHI ALARM SP DeltaV -> PLC"
  F26:132  PT_7010_LL_SP_DV  "PT-7010 LOLO ALARM SP DeltaV -> PLC"
  F26:133  PT_7010_HH_SP_DV  "PT-7010 HIHI ALARM SP DeltaV -> PLC"
  F26:134  PT_7020_LL_SP_DV  "PT-7020 LOLO ALARM SP DeltaV -> PLC"
  F26:135  PT_7020_HH_SP_DV  "PT-7020 HIHI ALARM SP DeltaV -> PLC"
  F26:136  FT_7000_LL_SP_DV  "FT-7000 LOLO ALARM SP DeltaV -> PLC"
  F26:137  FT_7000_HH_SP_DV  "FT-7000 HIHI ALARM SP DeltaV -> PLC"
  F26:138  FT_7005_LL_SP_DV  "FT-7005 LOLO ALARM SP DeltaV -> PLC"
  F26:139  FT_7005_HH_SP_DV  "FT-7005 HIHI ALARM SP DeltaV -> PLC"
  F26:140  FT_7008_LL_SP_DV  "FT-7008 LOLO ALARM SP DeltaV -> PLC"
  F26:141  FT_7008_HH_SP_DV  "FT-7008 HIHI ALARM SP DeltaV -> PLC"
  F26:142  FT_7025_LL_SP_DV  "FT-7025 LOLO ALARM SP DeltaV -> PLC"
  F26:143  FT_7025_HH_SP_DV  "FT-7025 HIHI ALARM SP DeltaV -> PLC"
  F26:144  FT_7050_LL_SP_DV  "FT-7050 LOLO ALARM SP DeltaV -> PLC"
  F26:145  FT_7050_HH_SP_DV  "FT-7050 HIHI ALARM SP DeltaV -> PLC"
  F26:146  LT_7050_LL_SP_DV  "LT-7050 LOLO ALARM SP DeltaV -> PLC"
  F26:147  LT_7050_HH_SP_DV  "LT-7050 HIHI ALARM SP DeltaV -> PLC"
  F26:148  PT_7000_LL_SP_DV  "PT-7000 LOLO ALARM SP DeltaV -> PLC"
  F26:149  PT_7000_HH_SP_DV  "PT-7000 HIHI ALARM SP DeltaV -> PLC"
  F26:150  PT_7015_LL_SP_DV  "PT-7015 LOLO ALARM SP DeltaV -> PLC"
  F26:151  PT_7015_HH_SP_DV  "PT-7015 HIHI ALARM SP DeltaV -> PLC"
  F26:152  PT_7025_LL_SP_DV  "PT-7025 LOLO ALARM SP DeltaV -> PLC"
  F26:153  PT_7025_HH_SP_DV  "PT-7025 HIHI ALARM SP DeltaV -> PLC"
  F26:154  FT_7030_LL_SP_DV  "FT-7030 LOLO ALARM SP DeltaV -> PLC"
  F26:155  FT_7030_HH_SP_DV  "FT-7030 HIHI ALARM SP DeltaV -> PLC"
  F26:156  FT_7040_LL_SP_DV  "FT-7040 LOLO ALARM SP DeltaV -> PLC"
  F26:157  FT_7040_HH_SP_DV  "FT-7040 HIHI ALARM SP DeltaV -> PLC"
  F26:158  FT_7052_LL_SP_DV  "FT-7052 LOLO ALARM SP DeltaV -> PLC"
  F26:159  FT_7052_HH_SP_DV  "FT-7052 HIHI ALARM SP DeltaV -> PLC"
  F26:160  LT_7030_LL_SP_DV  "LT-7030 LOLO ALARM SP DeltaV -> PLC"
  F26:161  LT_7030_HH_SP_DV  "LT-7030 HIHI ALARM SP DeltaV -> PLC"
  F26:162  PDT_7040_LL_SP_DV  "PDT-7040 LOLO ALARM SP DeltaV -> PLC"
  F26:163  PDT_7040_HH_SP_DV  "PDT-7040 HIHI ALARM SP DeltaV -> PLC"
  F26:164  PT_7030_LL_SP_DV  "PT-7030 LOLO ALARM SP DeltaV -> PLC"
  F26:165  PT_7030_HH_SP_DV  "PT-7030 HIHI ALARM SP DeltaV -> PLC"
  F26:166  PT_7040_LL_SP_DV  "PT-7040 LOLO ALARM SP DeltaV -> PLC"
  F26:167  PT_7040_HH_SP_DV  "PT-7040 HIHI ALARM SP DeltaV -> PLC"
  F26:168  PT_7050_LL_SP_DV  "PT-7050 LOLO ALARM SP DeltaV -> PLC"
  F26:169  PT_7050_HH_SP_DV  "PT-7050 HIHI ALARM SP DeltaV -> PLC"
  F26:170  ST_7040_LL_SP_DV  "ST-7040 LOLO ALARM SP DeltaV -> PLC"
  F26:171  ST_7040_HH_SP_DV  "ST-7040 HIHI ALARM SP DeltaV -> PLC"
  F26:172  FT_7095_LL_SP_DV  "FT-7095 LOLO ALARM SP DeltaV -> PLC"
  F26:173  FT_7095_HH_SP_DV  "FT-7095 HIHI ALARM SP DeltaV -> PLC"
  F26:174  FT_7110_LL_SP_DV  "FT-7110 LOLO ALARM SP DeltaV -> PLC"
  F26:175  FT_7110_HH_SP_DV  "FT-7110 HIHI ALARM SP DeltaV -> PLC"
  F26:176  FT_7130_LL_SP_DV  "FT-7130 LOLO ALARM SP DeltaV -> PLC"
  F26:177  FT_7130_HH_SP_DV  "FT-7130 HIHI ALARM SP DeltaV -> PLC"
  F26:178  FT_7132_LL_SP_DV  "FT-7132 LOLO ALARM SP DeltaV -> PLC"
  F26:179  FT_7132_HH_SP_DV  "FT-7132 HIHI ALARM SP DeltaV -> PLC"
  F26:180  FT_7145_LL_SP_DV  "FT-7145 LOLO ALARM SP DeltaV -> PLC"
  F26:181  FT_7145_HH_SP_DV  "FT-7145 HIHI ALARM SP DeltaV -> PLC"
  F26:182  LT_7110_LL_SP_DV  "LT-7110 LOLO ALARM SP DeltaV -> PLC"
  F26:183  LT_7110_HH_SP_DV  "LT-7110 HIHI ALARM SP DeltaV -> PLC"
  F26:184  LT_7130_LL_SP_DV  "LT-7130 LOLO ALARM SP DeltaV -> PLC"
  F26:185  LT_7130_HH_SP_DV  "LT-7130 HIHI ALARM SP DeltaV -> PLC"
  F26:186  PDT_7110_LL_SP_DV  "PDT-7110 LOLO ALARM SP DeltaV -> PLC"
  F26:187  PDT_7110_HH_SP_DV  "PDT-7110 HIHI ALARM SP DeltaV -> PLC"
  F26:188  PT_7110_LL_SP_DV  "PT-7110 LOLO ALARM SP DeltaV -> PLC"
  F26:189  PT_7110_HH_SP_DV  "PT-7110 HIHI ALARM SP DeltaV -> PLC"
  F26:190  PT_7111_LL_SP_DV  "PT-7111 LOLO ALARM SP DeltaV -> PLC"
  F26:191  PT_7111_HH_SP_DV  "PT-7111 HIHI ALARM SP DeltaV -> PLC"
  F26:192  PT_7130_LL_SP_DV  "PT-7130 LOLO ALARM SP DeltaV -> PLC"
  F26:193  PT_7130_HH_SP_DV  "PT-7130 HIHI ALARM SP DeltaV -> PLC"
  F26:194  ST_7110_LL_SP_DV  "ST-7110 LOLO ALARM SP DeltaV -> PLC"
  F26:195  ST_7110_HH_SP_DV  "ST-7110 HIHI ALARM SP DeltaV -> PLC"
  F26:196  ST_7130_LL_SP_DV  "ST-7130 LOLO ALARM SP DeltaV -> PLC"
  F26:197  ST_7130_HH_SP_DV  "ST-7130 HIHI ALARM SP DeltaV -> PLC"
  F26:198  FT_7120_LL_SP_DV  "FT-7120 LOLO ALARM SP DeltaV -> PLC"
  F26:199  FT_7120_HH_SP_DV  "FT-7120 HIHI ALARM SP DeltaV -> PLC"
  F26:200  FT_7140_LL_SP_DV  "FT-7140 LOLO ALARM SP DeltaV -> PLC"
  F26:201  FT_7140_HH_SP_DV  "FT-7140 HIHI ALARM SP DeltaV -> PLC"
  F26:202  TT_7009_LL_SP_DV  "TT-7009 LOLO ALARM SP DeltaV -> PLC"
  F26:203  TT_7009_HH_SP_DV  "TT-7009 HIHI ALARM SP DeltaV -> PLC"
  F26:204  TT_7010_LL_SP_DV  "TT-7010 LOLO ALARM SP DeltaV -> PLC"
  F26:205  TT_7010_HH_SP_DV  "TT-7010 HIHI ALARM SP DeltaV -> PLC"
  F26:206  TT_7020_LL_SP_DV  "TT-7020 LOLO ALARM SP DeltaV -> PLC"
  F26:207  TT_7020_HH_SP_DV  "TT-7020 HIHI ALARM SP DeltaV -> PLC"
  F26:208  TT_7000_LL_SP_DV  "TT-7000 LOLO ALARM SP DeltaV -> PLC"
  F26:209  TT_7000_HH_SP_DV  "TT-7000 HIHI ALARM SP DeltaV -> PLC"
  F26:210  TT_7015_LL_SP_DV  "TT-7015 LOLO ALARM SP DeltaV -> PLC"
  F26:211  TT_7015_HH_SP_DV  "TT-7015 HIHI ALARM SP DeltaV -> PLC"
  F26:212  TT_7025_LL_SP_DV  "TT-7025 LOLO ALARM SP DeltaV -> PLC"
  F26:213  TT_7025_HH_SP_DV  "TT-7025 HIHI ALARM SP DeltaV -> PLC"
  F26:214  TT_7026_LL_SP_DV  "TT-7026 LOLO ALARM SP DeltaV -> PLC"
  F26:215  TT_7026_HH_SP_DV  "TT-7026 HIHI ALARM SP DeltaV -> PLC"
  F26:216  TT_7050_LL_SP_DV  "TT-7050 LOLO ALARM SP DeltaV -> PLC"
  F26:217  TT_7050_HH_SP_DV  "TT-7050 HIHI ALARM SP DeltaV -> PLC"
  F26:218  TT_7030_LL_SP_DV  "TT-7030 LOLO ALARM SP DeltaV -> PLC"
  F26:219  TT_7030_HH_SP_DV  "TT-7030 HIHI ALARM SP DeltaV -> PLC"
  F26:220  TT_7040_LL_SP_DV  "TT-7040 LOLO ALARM SP DeltaV -> PLC"
  F26:221  TT_7040_HH_SP_DV  "TT-7040 HIHI ALARM SP DeltaV -> PLC"
  F26:222  TT_7042_LL_SP_DV  "TT-7042 LOLO ALARM SP DeltaV -> PLC"
  F26:223  TT_7042_HH_SP_DV  "TT-7042 HIHI ALARM SP DeltaV -> PLC"
  F26:224  TT_7043_LL_SP_DV  "TT-7043L LOLO ALARM SP DeltaV -> PLC"
  F26:225  TT_7043_HH_SP_DV  "TT-7043L HIHI ALARM SP DeltaV -> PLC"
  F26:226  TT_7044_LL_SP_DV  "TT-7043R LOLO ALARM SP DeltaV -> PLC"
  F26:227  TT_7044_HH_SP_DV  "TT-7043R HIHI ALARM SP DeltaV -> PLC"
  F26:228  TT_7045_LL_SP_DV  "TT-7045 LOLO ALARM SP DeltaV -> PLC"
  F26:229  TT_7045_HH_SP_DV  "TT-7045 HIHI ALARM SP DeltaV -> PLC"
  F26:230  TT_7046_LL_SP_DV  "TT-7046 LOLO ALARM SP DeltaV -> PLC"
  F26:231  TT_7046_HH_SP_DV  "TT-7046 HIHI ALARM SP DeltaV -> PLC"
  F26:232  TT_7047_LL_SP_DV  "TT-7047 LOLO ALARM SP DeltaV -> PLC"
  F26:233  TT_7047_HH_SP_DV  "TT-7047 HIHI ALARM SP DeltaV -> PLC"
  F26:234  TT_7110_LL_SP_DV  "TT-7110 LOLO ALARM SP DeltaV -> PLC"
  F26:235  TT_7110_HH_SP_DV  "TT-7110 HIHI ALARM SP DeltaV -> PLC"
  F26:236  TT_7111_LL_SP_DV  "TT-7111 LOLO ALARM SP DeltaV -> PLC"
  F26:237  TT_7111_HH_SP_DV  "TT-7111 HIHI ALARM SP DeltaV -> PLC"
  F26:238  TT_7118_LL_SP_DV  "TT-7118 LOLO ALARM SP DeltaV -> PLC"
  F26:239  TT_7118_HH_SP_DV  "TT-7118 HIHI ALARM SP DeltaV -> PLC"
  F26:240  TT_7119_LL_SP_DV  "TT-7119 LOLO ALARM SP DeltaV -> PLC"
  F26:241  TT_7119_HH_SP_DV  "TT-7119 HIHI ALARM SP DeltaV -> PLC"
  F26:242  TT_7130_LL_SP_DV  "TT-7130 LOLO ALARM SP DeltaV -> PLC"
  F26:243  TT_7130_HH_SP_DV  "TT-7130 HIHI ALARM SP DeltaV -> PLC"
  F26:244  ST_7010_H_AL_SP_DV  "FT-7140 HI ALARM SP DeltaV -> PLC"
  F26:245  ST_7010_HH_SP_DV  "ST-7010 HIHI ALARM SP DeltaV -> PLC"
  F26:246  TT_7135_LL_SP_DV  "TT-7135 LOLO ALARM SP DeltaV -> PLC"
  F26:247  TT_7135_HH_SP_DV  "TT-7135 HIHI ALARM SP DeltaV -> PLC"
  F26:248  TT_7140_LL_SP_DV  "TT-7140 LOLO ALARM SP DeltaV -> PLC"
  F26:249  TT_7140_HH_SP_DV  "TT-7140 HIHI ALARM SP DeltaV -> PLC"
  F26:250  TT_7145_LL_SP_DV  "TT-7145 LOLO ALARM SP DeltaV -> PLC"
  F26:251  TT_7145_HH_SP_DV  "TT-7145 HIHI ALARM SP DeltaV -> PLC"
  F26:252  PT_7026_HH_SP_DV  "PT-7026 HIHI ALARM SP DeltaV -> PLC"
  F26:253  PT_7026_H_AL_SP_DV  "PT-7026 HI ALARM SP DeltaV -> PLC"
  F26:254  PT_7026_L_AL_SP_DV  "PT-7026 LO ALARM SP DeltaV -> PLC"
  F26:255  PT_7026_LL_SP_DV  "PT-7026 LOLO ALARM SP DeltaV -> PLC"
  F27:0  TT_7027_HH_SP_DV  "TT-7027 HIHI ALARM SP DeltaV -> PLC"
  F27:1  TT_7027_H_AL_SP_DV  "TT-7027 HI ALARM SP DeltaV -> PLC"
  F27:2  TT_7027_L_AL_SP_DV  "TT-7027 LO ALARM SP DeltaV -> PLC"
  F27:3  TT_7027_LL_SP_DV  "TT-7027 LOLO ALARM SP DeltaV -> PLC"
  F27:4  FIC7015_KC_DV  "FIC7015 Kc DeltaV -> PLC"
  F27:5  FIC7015_TI_DV  "FIC7015 Ti DeltaV -> PLC"
  F27:6  FIC7015_TD_DV  "FIC7015 Td DeltaV -> PLC"
  F27:7  TIC7010_KC_DV  "TIC7010 Kc DeltaV -> PLC"
  F27:8  TIC7010_TI_DV  "TIC7010 Ti DeltaV -> PLC"
  F27:9  TIC7010_TD_DV  "TIC7010_Td DeltaV -> PLC"
  F27:10  FIC7000_KC_DV  "FIC7000 Kc DeltaV -> PLC"
  F27:11  FIC7000_TI_DV  "FIC7000 Ti DeltaV -> PLC"
  F27:12  FIC7000_TD_DV  "FIC7000 Td DeltaV -> PLC"
  F27:13  FIC7005_KC_DV  "FIC7005 Kc DeltaV -> PLC"
  F27:14  FIC7005_TI_DV  "FIC7005 Ti DeltaV -> PLC"
  F27:15  FIC7005_TD_DV  "FIC7005 Td DeltaV -> PLC"
  F27:16  FIC7008_KC_DV  "FIC7008 Kc DeltaV -> PLC"
  F27:17  FIC7008_TI_DV  "FIC7008 Ti DeltaV -> PLC"
  F27:18  FIC7008_TD_DV  "FIC7008 Td DeltaV -> PLC"
  F27:19  FIC7010_KC_DV  "FIC7010 Kc DeltaV -> PLC"
  F27:20  FIC7010_TI_DV  "FIC7010 Ti DeltaV -> PLC"
  F27:21  FIC7010_TD_DV  "FIC7010_Td DeltaV -> PLC"
  F27:22  LIC7050_KC_DV  "LIC7050 Kc DeltaV -> PLC"
  F27:23  LIC7050_TI_DV  "LIC7050 Ti DeltaV -> PLC"
  F27:24  LIC7050_TD_DV  "LIC7050 Td DeltaV -> PLC"
  F27:25  TIC7026_KC_DV  "TIC7026 Kc DeltaV -> PLC"
  F27:26  TIC7026_TI_DV  "TIC7026 Ti DeltaV -> PLC"
  F27:27  TIC7026_TD_DV  "TIC7026 Td DeltaV -> PLC"
  F27:28  FIC7030_KC_DV  "FIC7030 Kc DeltaV -> PLC"
  F27:29  FIC7030_TI_DV  "FIC7030 Ti DeltaV -> PLC"
  F27:30  FIC7030_TD_DV  "FIC7030 Td DeltaV -> PLC"
  F27:31  FIC7040_KC_DV  "FIC7040 Kc DeltaV -> PLC"
  F27:32  FIC7040_TI_DV  "FIC7040 Ti DeltaV -> PLC"
  F27:33  FIC7040_TD_DV  "FIC7040 Td DeltaV -> PLC"
  F27:34  LIC7030_KC_DV  "LIC7030 Kc DeltaV -> PLC"
  F27:35  LIC7030_TI_DV  "LIC7030 Ti DeltaV -> PLC"
  F27:36  LIC7030_TD_DV  "LIC7030 Td DeltaV -> PLC"
  F27:37  PIC7050_KC_DV  "PIC7050 Kc DeltaV -> PLC"
  F27:38  PIC7050_TI_DV  "PIC7050 Ti DeltaV -> PLC"
  F27:39  PIC7050_TD_DV  "PIC7050 Td DeltaV -> PLC"
  F27:40  TIC7047_KC_DV  "TIC7047 Kc DeltaV -> PLC"
  F27:41  TIC7047_TI_DV  "TIC7047 Ti DeltaV -> PLC"
  F27:42  TIC7047_TD_DV  "TIC7047 Td DeltaV -> PLC"
  F27:43  TIC7045_KC_DV  "TIC7045 Kc DeltaV -> PLC"
  F27:44  TIC7045_TI_DV  "TIC7045 Ti DeltaV -> PLC"
  F27:45  TIC7045_TD_DV  "TIC7045 Td DeltaV -> PLC"
  F27:46  FIC7110_KC_DV  "FIC7110 Kc DeltaV -> PLC"
  F27:47  FIC7110_TI_DV  "FIC7110 Ti DeltaV -> PLC"
  F27:48  FIC7110_TD_DV  "FIC7110 Td DeltaV -> PLC"
  F27:49  LIC7110_KC_DV  "LIC7110 Kc DeltaV -> PLC"
  F27:50  LIC7110_TI_DV  "LIC7110 Ti DeltaV -> PLC"
  F27:51  LIC7110_TD_DV  "LIC7110 Td DeltaV -> PLC"
  F27:52  LIC7130_KC_DV  "LIC7130 Kc DeltaV -> PLC"
  F27:53  LIC7130_TI_DV  "LIC7130 Ti DeltaV -> PLC"
  F27:54  LIC7130_TD_DV  "LIC7130 Td DeltaV -> PLC"
  F27:55  PIC7130_KC_DV  "PIC7130 Kc DeltaV -> PLC"
  F27:56  PIC7130_TI_DV  "PIC7130 Ti DeltaV -> PLC"
  F27:57  PIC7130_TD_DV  "PIC7130 Td DeltaV -> PLC"
  F27:58  TIC7110_KC_DV  "TIC7110 Kc DeltaV -> PLC"
  F27:59  TIC7110_TI_DV  "TIC7110 Ti DeltaV -> PLC"
  F27:60  TIC7110_TD_DV  "TIC7110 Td DeltaV -> PLC"
  F27:61  FIC7140_KC_DV  "FIC7140 Kc DeltaV -> PLC"
  F27:62  FIC7140_TI_DV  "FIC7140 Ti DeltaV -> PLC"
  F27:63  FIC7140_TD_DV  "FIC7140 Td DeltaV -> PLC"
  F27:64  TIC7010_SP_DV  "TIC7010 SP DeltaV -> PLC"
  F27:65  FIC7015_SP_DV  "FIC7015 SP DeltaV -> PLC"
  F27:66  FIC7015_OP_DV  "FIC7015 OP DeltaV -> PLC"
  F27:67  TIC7010_OP_DV  "TIC7010 OP DeltaV -> PLC"
  F27:68  FIC7000_SP_DV  "FIC7000 SP DeltaV -> PLC"
  F27:69  FIC7000_OP_DV  "FIC7000 OP DeltaV -> PLC"
  F27:70  FIC7005_SP_DV  "FIC7005 SP DeltaV -> PLC"
  F27:71  FIC7005_OP_DV  "FIC7005 OP DeltaV -> PLC"
  F27:72  FIC7008_SP_DV  "FIC7008 SP DeltaV -> PLC"
  F27:73  FIC7008_OP_DV  "FIC7008 OP DeltaV -> PLC"
  F27:74  FIC7010_SP_DV  "FIC7010 SP DeltaV -> PLC"
  F27:75  FIC7010_OP_DV  "FIC7010 OP DeltaV -> PLC"
  F27:76  LIC7050_SP_DV  "LIC7050 SP DeltaV -> PLC"
  F27:77  LIC7050_OP_DV  "LIC7050 OP DeltaV -> PLC"
  F27:78  TIC7026_SP_DV  "TIC7026 SP DeltaV -> PLC"
  F27:79  TIC7026_OP_DV  "TIC7026 OP DeltaV -> PLC"
  F27:80  FIC7030_SP_DV  "FIC7030 SP DeltaV -> PLC"
  F27:81  FIC7030_OP_DV  "FIC7030 OP DeltaV -> PLC"
  F27:82  FIC7040_SP_DV  "FIC7040 SP DeltaV -> PLC"
  F27:83  FIC7040_OP_DV  "FIC7040 OP DeltaV -> PLC"
  F27:84  LIC7030_OP_DV  "LIC7030 OP DeltaV -> PLC"
  F27:85  PIC7050_OP_DV  "PIC7050 OP DeltaV -> PLC"
  F27:86  TIC7047_SP_DV  "TIC7047 SP DeltaV -> PLC"
  F27:87  TIC7047_OP_DV  "TIC7047 OP DeltaV -> PLC"
  F27:88  TIC7045_SP_DV  "TIC7045 SP DeltaV -> PLC"
  F27:89  TIC7045_OP_DV  "TIC7045 OP DeltaV -> PLC"
  F27:90  FIC7110_SP_DV  "FIC7110 SP DeltaV -> PLC"
  F27:91  FIC7110_OP_DV  "FIC7110 OP DeltaV -> PLC"
  F27:92  LIC7110_SP_DV  "LIC7110 SP DeltaV -> PLC"
  F27:93  LIC7110_OP_DV  "LIC7110 OP DeltaV -> PLC"
  F27:94  LIC7130_SP_DV  "LIC7130 SP DeltaV -> PLC"
  F27:95  LIC7130_OP_DV  "LIC7130 OP DeltaV -> PLC"
  F27:96  PIC7130_SP_DV  "PIC7130 SP DeltaV -> PLC"
  F27:97  PIC7130_OP_DV  "PIC7130 OP DeltaV -> PLC"
  F27:98  TIC7110_SP_DV  "TIC7110 SP DeltaV -> PLC"
  F27:99  TIC7110_OP_DV  "TIC7110 OP DeltaV -> PLC"
  F27:100  FIC7140_SP_DV  "FIC7140 SP DeltaV -> PLC"
  F27:101  FIC7140_OP_DV  "FIC7140 OP DeltaV -> PLC"
  F27:102  F7002_L_AL_DLY_SP_DV  "FT-7002 LO ALM DLY SP DeltaV -> PLC"
  F27:103  F7002_H_AL_DLY_SP_DV  "FT-7002 HI ALM DLY SP DeltaV -> PLC"
  F27:104  F7010_L_AL_DLY_SP_DV  "FT-7010 LO ALM DLY SP DeltaV -> PLC"
  F27:105  F7010_H_AL_DLY_SP_DV  "FT-7010 HI ALM DLY SP DeltaV -> PLC"
  F27:106  L7010_L_AL_DLY_SP_DV  "LT-7010 LO ALM DLY SP DeltaV -> PLC"
  F27:107  L7010_H_AL_DLY_SP_DV  "LT-7010 HI ALM DLY SP DeltaV -> PLC"
  F27:108  P7010_L_AL_DLY_SP_DV  "PT-7010 LO ALM DLY SP DeltaV -> PLC"
  F27:109  P7010_H_AL_DLY_SP_DV  "PT-7010 HI ALM DLY SP DeltaV -> PLC"
  F27:110  P7020_L_AL_DLY_SP_DV  "PT-7020 LO ALM DLY SP DeltaV -> PLC"
  F27:111  P7020_H_AL_DLY_SP_DV  "PT-7020 HI ALM DLY SP DeltaV -> PLC"
  F27:112  F7000_L_AL_DLY_SP_DV  "FT-7000 LO ALM DLY SP DeltaV -> PLC"
  F27:113  F7000_H_AL_DLY_SP_DV  "FT-7000 HI ALM DLY SP DeltaV -> PLC"
  F27:114  F7005_L_AL_DLY_SP_DV  "FT-7005 LO ALM DLY SP DeltaV -> PLC"
  F27:115  F7005_H_AL_DLY_SP_DV  "FT-7005 HI ALM DLY SP DeltaV -> PLC"
  F27:116  F7008_L_AL_DLY_SP_DV  "FT-7008 LO ALM DLY SP DeltaV -> PLC"
  F27:117  F7008_H_AL_DLY_SP_DV  "FT-7008 HI ALM DLY SP DeltaV -> PLC"
  F27:118  F7025_L_AL_DLY_SP_DV  "FT-7025 LO ALM DLY SP DeltaV -> PLC"
  F27:119  F7025_H_AL_DLY_SP_DV  "FT-7025 HI ALM DLY SP DeltaV -> PLC"
  F27:120  F7050_L_AL_DLY_SP_DV  "FT-7050 LO ALM DLY SP DeltaV -> PLC"
  F27:121  F7050_H_AL_DLY_SP_DV  "FT-7050 HI ALM DLY SP DeltaV -> PLC"
  F27:122  L7050_L_AL_DLY_SP_DV  "LT-7050 LO ALM DLY SP DeltaV -> PLC"
  F27:123  L7050_H_AL_DLY_SP_DV  "LT-7050 HI ALM DLY SP DeltaV -> PLC"
  F27:124  P7000_L_AL_DLY_SP_DV  "PT-7000 LO ALM DLY SP DeltaV -> PLC"
  F27:125  P7000_H_AL_DLY_SP_DV  "PT-7000 HI ALM DLY SP DeltaV -> PLC"
  F27:126  P7015_L_AL_DLY_SP_DV  "PT-7015 LO ALM DLY SP DeltaV -> PLC"
  F27:127  P7015_H_AL_DLY_SP_DV  "PT-7015 HI ALM DLY SP DeltaV -> PLC"
  F27:128  P7025_L_AL_DLY_SP_DV  "PT-7025 LO ALM DLY SP DeltaV -> PLC"
  F27:129  P7025_H_AL_DLY_SP_DV  "PT-7025 HI ALM DLY SP DeltaV -> PLC"
  F27:130  F7030_L_AL_DLY_SP_DV  "FT-7030 LO ALM DLY SP DeltaV -> PLC"
  F27:131  F7030_H_AL_DLY_SP_DV  "FT-7030 HI ALM DLY SP DeltaV -> PLC"
  F27:132  F7040_L_AL_DLY_SP_DV  "FT-7040 LO ALM DLY SP DeltaV -> PLC"
  F27:133  F7040_H_AL_DLY_SP_DV  "FT-7040 HI ALM DLY SP DeltaV -> PLC"
  F27:134  F7052_L_AL_DLY_SP_DV  "FT-7052 LO ALM DLY SP DeltaV -> PLC"
  F27:135  F7052_H_AL_DLY_SP_DV  "FT-7052 HI ALM DLY SP DeltaV -> PLC"
  F27:136  L7030_L_AL_DLY_SP_DV  "LT-7030 LO ALM DLY SP DeltaV -> PLC"
  F27:137  L7030_H_AL_DLY_SP_DV  "LT-7030 HI ALM DLY SP DeltaV -> PLC"
  F27:138  PD7040_L_AL_D_SP_DV  "PDT-7040 LO ALM DLY SP DeltaV -> PLC"
  F27:139  PD7040_H_AL_D_SP_DV  "PDT-7040 HI ALM DLY SP DeltaV -> PLC"
  F27:140  P7030_L_AL_DLY_SP_DV  "PT-7030 LO ALM DLY SP DeltaV -> PLC"
  F27:141  P7030_H_AL_DLY_SP_DV  "PT-7030 HI ALM DLY SP DeltaV -> PLC"
  F27:142  P7040_L_AL_DLY_SP_DV  "PT-7040 LO ALM DLY SP DeltaV -> PLC"
  F27:143  P7040_H_AL_DLY_SP_DV  "PT-7040 HI ALM DLY SP DeltaV -> PLC"
  F27:144  P7050_L_AL_DLY_SP_DV  "PT-7050 LO ALM DLY SP DeltaV -> PLC"
  F27:145  P7050_H_AL_DLY_SP_DV  "PT-7050 HI ALM DLY SP DeltaV -> PLC"
  F27:146  S7040_L_AL_DLY_SP_DV  "ST-7040 LO ALM DLY SP DeltaV -> PLC"
  F27:147  S7040_H_AL_DLY_SP_DV  "ST-7040 HI ALM DLY SP DeltaV -> PLC"
  F27:148  F7095_L_AL_DLY_SP_DV  "FT-7095 LO ALM DLY SP DeltaV -> PLC"
  F27:149  F7095_H_AL_DLY_SP_DV  "FT-7095 HI ALM DLY SP DeltaV -> PLC"
  F27:150  F7110_L_AL_DLY_SP_DV  "FT-7110 LO ALM DLY SP DeltaV -> PLC"
  F27:151  F7110_H_AL_DLY_SP_DV  "FT-7110 HI ALM DLY SP DeltaV -> PLC"
  F27:152  F7130_L_AL_DLY_SP_DV  "FT-7130 LO ALM DLY SP DeltaV -> PLC"
  F27:153  F7130_H_AL_DLY_SP_DV  "FT-7130 HI ALM DLY SP DeltaV -> PLC"
  F27:154  F7132_L_AL_DLY_SP_DV  "FT-7132 LO ALM DLY SP DeltaV -> PLC"
  F27:155  F7132_H_AL_DLY_SP_DV  "FT-7132 HI ALM DLY SP DeltaV -> PLC"
  F27:156  F7145_L_AL_DLY_SP_DV  "FT-7145 LO ALM DLY SP DeltaV -> PLC"
  F27:157  F7145_H_AL_DLY_SP_DV  "FT-7145 HI ALM DLY SP DeltaV -> PLC"
  F27:158  L7110_L_AL_DLY_SP_DV  "LT-7110 LO ALM DLY SP DeltaV -> PLC"
  F27:159  L7110_H_AL_DLY_SP_DV  "LT-7110 HI ALM DLY SP DeltaV -> PLC"
  F27:160  L7130_L_AL_DLY_SP_DV  "LT-7130 LO ALM DLY SP DeltaV -> PLC"
  F27:161  L7130_H_AL_DLY_SP_DV  "LT-7130 HI ALM DLY SP DeltaV -> PLC"
  F27:162  PD7110_L_AL_D_SP_DV  "PDT-7110 LO ALM DLY SP DeltaV -> PLC"
  F27:163  PD7110_H_AL_D_SP_DV  "PDT-7110 HI ALM DLY SP DeltaV -> PLC"
  F27:164  P7110_L_AL_DLY_SP_DV  "PT-7110 LO ALM DLY SP DeltaV -> PLC"
  F27:165  P7110_H_AL_DLY_SP_DV  "PT-7110 HI ALM DLY SP DeltaV -> PLC"
  F27:166  P7111_L_AL_DLY_SP_DV  "PT-7111 LO ALM DLY SP DeltaV -> PLC"
  F27:167  P7111_H_AL_DLY_SP_DV  "PT-7111 HI ALM DLY SP DeltaV -> PLC"
  F27:168  P7130_L_AL_DLY_SP_DV  "PT-7130 LO ALM DLY SP DeltaV -> PLC"
  F27:169  P7130_H_AL_DLY_SP_DV  "PT-7130 HI ALM DLY SP DeltaV -> PLC"
  F27:170  S7110_L_AL_DLY_SP_DV  "ST-7110 LO ALM DLY SP DeltaV -> PLC"
  F27:171  S7110_H_AL_DLY_SP_DV  "ST-7110 HI ALM DLY SP DeltaV -> PLC"
  F27:172  S7130_L_AL_DLY_SP_DV  "ST-7130 LO ALM DLY SP DeltaV -> PLC"
  F27:173  S7130_H_AL_DLY_SP_DV  "ST-7130 HI ALM DLY SP DeltaV -> PLC"
  F27:174  F7120_L_AL_DLY_SP_DV  "FT-7120 LO ALM DLY SP DeltaV -> PLC"
  F27:175  F7120_H_AL_DLY_SP_DV  "FT-7120 HI ALM DLY SP DeltaV -> PLC"
  F27:176  F7140_L_AL_DLY_SP_DV  "FT-7140 LO ALM DLY SP DeltaV -> PLC"
  F27:177  F7140_H_AL_DLY_SP_DV  "FT-7140 HI ALM DLY SP DeltaV -> PLC"
  F27:178  T7009_L_AL_DLY_SP_DV  "TT-7009 LO ALM DLY SP DeltaV -> PLC"
  F27:179  T7009_H_AL_DLY_SP_DV  "TT-7009 HI ALM DLY SP DeltaV -> PLC"
  F27:180  T7010_L_AL_DLY_SP_DV  "TT-7010 LO ALM DLY SP DeltaV -> PLC"
  F27:181  T7010_H_AL_DLY_SP_DV  "TT-7010 HI ALM DLY SP DeltaV -> PLC"
  F27:182  T7020_L_AL_DLY_SP_DV  "TT-7020 LO ALM DLY SP DeltaV -> PLC"
  F27:183  T7020_H_AL_DLY_SP_DV  "TT-7020 HI ALM DLY SP DeltaV -> PLC"
  F27:184  T7000_L_AL_DLY_SP_DV  "TT-7000 LO ALM DLY SP DeltaV -> PLC"
  F27:185  T7000_H_AL_DLY_SP_DV  "TT-7000 HI ALM DLY SP DeltaV -> PLC"
  F27:186  T7015_L_AL_DLY_SP_DV  "TT-7015 LO ALM DLY SP DeltaV -> PLC"
  F27:187  T7015_H_AL_DLY_SP_DV  "TT-7015 HI ALM DLY SP DeltaV -> PLC"
  F27:188  T7025_L_AL_DLY_SP_DV  "TT-7025 LO ALM DLY SP DeltaV -> PLC"
  F27:189  T7025_H_AL_DLY_SP_DV  "TT-7025 HI ALM DLY SP DeltaV -> PLC"
  F27:190  T7026_L_AL_DLY_SP_DV  "TT-7026 LO ALM DLY SP DeltaV -> PLC"
  F27:191  T7026_H_AL_DLY_SP_DV  "TT-7026 HI ALM DLY SP DeltaV -> PLC"
  F27:192  T7050_L_AL_DLY_SP_DV  "TT-7050 LO ALM DLY SP DeltaV -> PLC"
  F27:193  T7050_H_AL_DLY_SP_DV  "TT-7050 HI ALM DLY SP DeltaV -> PLC"
  F27:194  T7030_L_AL_DLY_SP_DV  "TT-7030 LO ALM DLY SP DeltaV -> PLC"
  F27:195  T7030_H_AL_DLY_SP_DV  "TT-7030 HI ALM DLY SP DeltaV -> PLC"
  F27:196  T7040_L_AL_DLY_SP_DV  "TT-7040 LO ALM DLY SP DeltaV -> PLC"
  F27:197  T7040_H_AL_DLY_SP_DV  "TT-7040 HI ALM DLY SP DeltaV -> PLC"
  F27:198  T7042_L_AL_DLY_SP_DV  "TT-7042 LO ALM DLY SP DeltaV -> PLC"
  F27:199  T7042_H_AL_DLY_SP_DV  "TT-7042 HI ALM DLY SP DeltaV -> PLC"
  F27:200  T7043_LALM_DLY_SP_DV  "TT-7043 LO ALM DLY SP DeltaV -> PLC"
  F27:201  T7043_HALM_DLY_SP_DV  "TT-7043 HI ALM DLY SP DeltaV -> PLC"
  F27:202  T7044_LALM_DLY_SP_DV  "TT-7044 LO ALM DLY SP DeltaV -> PLC"
  F27:203  T7044_HALM_DLY_SP_DV  "TT-7044 HI ALM DLY SP DeltaV -> PLC"
  F27:204  T7045_L_AL_DLY_SP_DV  "TT-7045 LO ALM DLY SP DeltaV -> PLC"
  F27:205  T7045_H_AL_DLY_SP_DV  "TT-7045 HI ALM DLY SP DeltaV -> PLC"
  F27:206  T7046_L_AL_DLY_SP_DV  "TT-7046 LO ALM DLY SP DeltaV -> PLC"
  F27:207  T7046_H_AL_DLY_SP_DV  "TT-7046 HI ALM DLY SP DeltaV -> PLC"
  F27:208  T7047_L_AL_DLY_SP_DV  "TT-7047 LO ALM DLY SP DeltaV -> PLC"
  F27:209  T7047_H_AL_DLY_SP_DV  "TT-7047 HI ALM DLY SP DeltaV -> PLC"
  F27:210  T7110_L_AL_DLY_SP_DV  "TT-7110 LO ALM DLY SP DeltaV -> PLC"
  F27:211  T7110_H_AL_DLY_SP_DV  "TT-7110 HI ALM DLY SP DeltaV -> PLC"
  F27:212  T7111_L_AL_DLY_SP_DV  "TT-7111 LO ALM DLY SP DeltaV -> PLC"
  F27:213  T7111_H_AL_DLY_SP_DV  "TT-7111 HI ALM DLY SP DeltaV -> PLC"
  F27:214  T7118_L_AL_DLY_SP_DV  "TT-7118 LO ALM DLY SP DeltaV -> PLC"
  F27:215  T7118_H_AL_DLY_SP_DV  "TT-7118 HI ALM DLY SP DeltaV -> PLC"
  F27:216  T7119_L_AL_DLY_SP_DV  "TT-7119 LO ALM DLY SP DeltaV -> PLC"
  F27:217  T7119_H_AL_DLY_SP_DV  "TT-7119 HI ALM DLY SP DeltaV -> PLC"
  F27:218  T7130_L_AL_DLY_SP_DV  "TT-7130 LO ALM DLY SP DeltaV -> PLC"
  F27:219  T7130_H_AL_DLY_SP_DV  "TT-7130 HI ALM DLY SP DeltaV -> PLC"
  F27:220  S7010_LL_DLY_SP_DV  "ST-7010 LL ALM DLY SP DeltaV -> PLC"
  F27:221  S7010_HH_DLY_SP_DV  "ST-7010 HH ALM DLY SP DeltaV -> PLC"
  F27:222  T7135_L_AL_DLY_SP_DV  "TT-7135 LO ALM DLY SP DeltaV -> PLC"
  F27:223  T7135_H_AL_DLY_SP_DV  "TT-7135 HI ALM DLY SP DeltaV -> PLC"
  F27:224  T7140_L_AL_DLY_SP_DV  "TT-7140 LO ALM DLY SP DeltaV -> PLC"
  F27:225  T7140_H_AL_DLY_SP_DV  "TT-7140 HI ALM DLY SP DeltaV -> PLC"
  F27:226  T7145_L_AL_DLY_SP_DV  "TT-7145 LO ALM DLY SP DeltaV -> PLC"
  F27:227  T7145_H_AL_DLY_SP_DV  "TT-7145 HI ALM DLY SP DeltaV -> PLC"
  F27:228  F7002_LL_DLY_SP_DV  "FT-7002 LOLO ALM DLY SP DeltaV -> PLC"
  F27:229  F7002_HH_DLY_SP_DV  "FT-7002 HIHI ALM DLY SP DeltaV -> PLC"
  F27:230  F7010_LL_DLY_SP_DV  "FT-7010 LOLO ALM DLY SP DeltaV -> PLC"
  F27:231  F7010_HH_DLY_SP_DV  "FT-7010 HIHI ALM DLY SP DeltaV -> PLC"
  F27:232  L7010_LL_DLY_SP_DV  "LT-7010 LOLO ALM DLY SP DeltaV -> PLC"
  F27:233  L7010_HH_DLY_SP_DV  "LT-7010 HIHI ALM DLY SP DeltaV -> PLC"
  F27:234  P7010_LL_DLY_SP_DV  "PT-7010 LOLO ALM DLY SP DeltaV -> PLC"
  F27:235  P7010_HH_DLY_SP_DV  "PT-7010 HIHI ALM DLY SP DeltaV -> PLC"
  F27:236  P7020_LL_DLY_SP_DV  "PT-7020 LOLO ALM DLY SP DeltaV -> PLC"
  F27:237  P7020_HH_DLY_SP_DV  "PT-7020 HIHI ALM DLY SP DeltaV -> PLC"
  F27:238  F7000_LL_DLY_SP_DV  "FT-7000 LOLO ALM DLY SP DeltaV -> PLC"
  F27:239  F7000_HH_DLY_SP_DV  "FT-7000 HIHI ALM DLY SP DeltaV -> PLC"
  F27:240  F7005_LL_DLY_SP_DV  "FT-7005 LOLO ALM DLY SP DeltaV -> PLC"
  F27:241  F7005_HH_DLY_SP_DV  "FT-7005 HIHI ALM DLY SP DeltaV -> PLC"
  F27:242  F7008_LL_DLY_SP_DV  "FT-7008 LOLO ALM DLY SP DeltaV -> PLC"
  F27:243  F7008_HH_DLY_SP_DV  "FT-7008 HIHI ALM DLY SP DeltaV -> PLC"
  F27:244  F7025_LL_DLY_SP_DV  "FT-7025 LOLO ALM DLY SP DeltaV -> PLC"
  F27:245  F7025_HH_DLY_SP_DV  "FT-7025 HIHI ALM DLY SP DeltaV -> PLC"
  F27:246  F7050_LL_DLY_SP_DV  "FT-7050 LOLO ALM DLY SP DeltaV -> PLC"
  F27:247  F7050_HH_DLY_SP_DV  "FT-7050 HIHI ALM DLY SP DeltaV -> PLC"
  F27:248  L7050_LL_DLY_SP_DV  "LT-7050 LOLO ALM DLY SP DeltaV -> PLC"
  F27:249  L7050_HH_DLY_SP_DV  "LT-7050 HIHI ALM DLY SP DeltaV -> PLC"
  F27:250  P7000_LL_DLY_SP_DV  "PT-7000 LOLO ALM DLY SP DeltaV -> PLC"
  F27:251  P7000_HH_DLY_SP_DV  "PT-7000 HIHI ALM DLY SP DeltaV -> PLC"
  F27:252  P7015_LL_DLY_SP_DV  "PT-7015 LOLO ALM DLY SP DeltaV -> PLC"
  F27:253  P7015_HH_DLY_SP_DV  "PT-7015 HIHI ALM DLY SP DeltaV -> PLC"
  F27:254  P7025_LL_DLY_SP_DV  "PT-7025 LOLO ALM DLY SP DeltaV -> PLC"
  F27:255  P7025_HH_DLY_SP_DV  "PT-7025 HIHI ALM DLY SP DeltaV -> PLC"
  F28:0  F7030_LL_DLY_SP_DV  "FT-7030 LOLO ALM DLY SP DeltaV -> PLC"
  F28:1  F7030_HH_DLY_SP_DV  "FT-7030 HIHI ALM DLY SP DeltaV -> PLC"
  F28:2  F7040_LL_DLY_SP_DV  "FT-7040 LOLO ALM DLY SP DeltaV -> PLC"
  F28:3  F7040_HH_DLY_SP_DV  "FT-7040 HIHI ALM DLY SP DeltaV -> PLC"
  F28:4  F7052_LL_DLY_SP_DV  "FT-7052 LOLO ALM DLY SP DeltaV -> PLC"
  F28:5  F7052_HH_DLY_SP_DV  "FT-7052 HIHI ALM DLY SP DeltaV -> PLC"
  F28:6  L7030_LL_DLY_SP_DV  "LT-7030 LOLO ALM DLY SP DeltaV -> PLC"
  F28:7  L7030_HH_DLY_SP_DV  "LT-7030 HIHI ALM DLY SP DeltaV -> PLC"
  F28:8  PD7040_LL_DLY_SP_DV  "PDT-7040 LOLO ALM DLY SP DeltaV -> PLC"
